# B&R Automation Studio project NAINV104C00R8L515F00 (part 18)

#### Act_Background.st
```iecst
(** 2020-10-05 **)
ACTION Act_Background: //For Standard Machines

	IF EDGEPOS(p_bManual) THEN

		fbBlink(bEn := FALSE);
		fbWarning(bEn := FALSE);

		bTLRed		:= FALSE;
		bTLAmber	:= TRUE;
		bTLGreen	:= FALSE;
		bBuzBeep	:= FALSE;

	ELSIF p_bManual THEN

		IF p_bErr = TRUE THEN

			fbBlink.tOnTm	:= p_tTLErrBlinkTm; //Error T#500ms (from NtParam)
			fbBlink.tOffTm	:= p_tTLErrBlinkTm; //Error T#500ms (from NtParam)

			fbWarning.tOnTm					:= p_tBuzErrOnTm; //Warn T#500ms (from NtParam)
			fbWarning.tOffTm				:= p_tBuzErrOnTm; //Warn T#500ms (from NtParam)
			fbWarning.tRstTm				:= p_tBuzErrRestTm; //Rest 5 seconds (from NtParam)
			fbWarning.usiOnCnt				:= p_usiBuzErrOnCntr; //Count 3 times (from NtParam)
			fbWarning.bStopAftRptSeqEn		:= p_bBuzErrStopSeqEn; //Enable Sequence Count (from NtParam)
			fbWarning.usiStopAftRptSeqCntr	:= p_usiBuzErrStopSeqCntr; //Sequence Counter  (from NtParam)

			fbBlink(bEn := TRUE);
			fbWarning(bEn := TRUE);

			bTLRed		:= fbBlink.bOut;
			bBuzBeep	:= (fbWarning.bOut) AND (p_bMuteBuz = FALSE);

			bManualErrOn := TRUE;

		ELSIF bManualErrOn THEN

			fbBlink(bEn := FALSE);
			fbWarning(bEn := FALSE);

			bTLRed		:= FALSE;
			bBuzBeep	:= FALSE;

			bManualErrOn := FALSE;

		END_IF

	ELSIF p_bManual = FALSE THEN

		bManualErrOn := FALSE;

		IF p_bStartup = TRUE THEN

			fbBlink(bEn := FALSE);
			fbWarning(bEn := FALSE);

			bTLRed		:= TRUE;
			bTLAmber	:= TRUE;
			bTLGreen	:= TRUE;
			bBuzBeep	:= FALSE;

		ELSIF p_bErr = TRUE THEN

			fbBlink.tOnTm	:= p_tTLErrBlinkTm; //Error T#500ms (from NtParam)
			fbBlink.tOffTm	:= p_tTLErrBlinkTm; //Error T#500ms (from NtParam)

			fbWarning.tOnTm					:= p_tBuzErrOnTm; //Warn T#500ms (from NtParam)
			fbWarning.tOffTm				:= p_tBuzErrOnTm; //Warn T#500ms (from NtParam)
			fbWarning.tRstTm				:= p_tBuzErrRestTm; //Rest 5 seconds (from NtParam)
			fbWarning.usiOnCnt				:= p_usiBuzErrOnCntr; //Count 3 times (from NtParam)
			fbWarning.bStopAftRptSeqEn		:= p_bBuzErrStopSeqEn; //Enable Sequence Count (from NtParam)
			fbWarning.usiStopAftRptSeqCntr	:= p_usiBuzErrStopSeqCntr; //Sequence Counter  (from NtParam)

			fbBlink(bEn := TRUE);
			fbWarning(bEn := TRUE);

			bTLRed		:= fbBlink.bOut;
			bTLAmber	:= FALSE;
			bTLGreen	:= FALSE;
			bBuzBeep	:= (fbWarning.bOut) AND (p_bMuteBuz = FALSE);

		ELSIF p_bErrNoBuz = TRUE THEN

			fbBlink.tOnTm	:= p_tTLErrBlinkTm;
			fbBlink.tOffTm	:= p_tTLErrBlinkTm;
			fbBlink(bEn := TRUE);
			fbWarning(bEn := FALSE);

			bTLRed		:= fbBlink.bOut;
			bTLAmber	:= FALSE;
			bTLGreen	:= FALSE;
			bBuzBeep	:= FALSE;

		ELSIF p_bWarning = TRUE THEN

			fbBlink.tOnTm	:= p_tTLWarnBlinkTm; //Warn T#500ms (from NtParam)
			fbBlink.tOffTm	:= p_tTLWarnBlinkTm; //Warn T#500ms (from NtParam)

			fbWarning.tOnTm					:= p_tBuzWarnOnTm; //Warn T#500ms (from NtParam)
			fbWarning.tOffTm				:= p_tBuzWarnOnTm; //Warn T#500ms (from NtParam)
			fbWarning.tRstTm				:= p_tBuzWarnRestTm; //Rest 5 seconds (from NtParam)
			fbWarning.usiOnCnt				:= p_usiBuzWarnOnCntr; //Count 3 times (from NtParam)
			fbWarning.bStopAftRptSeqEn		:= p_bBuzWarnStopSeqEn; //Enable Sequence Count (from NtParam)
			fbWarning.usiStopAftRptSeqCntr	:= p_usiBuzWarnStopSeqCntr; //Sequence Counter  (from NtParam)

			fbBlink(bEn := TRUE);
			fbWarning(bEn := TRUE);

			bTLRed		:= p_bStandby;
			bTLAmber	:= fbBlink.bOut;
			bTLGreen	:= p_bOps;
			bBuzBeep	:= fbWarning.bOut AND (p_bMuteBuz = FALSE);

		ELSIF p_bWarningNoBuz = TRUE THEN

			fbBlink.tOnTm	:= p_tTLWarnBlinkTm;
			fbBlink.tOffTm	:= p_tTLWarnBlinkTm;
			fbBlink(bEn := TRUE);
			fbWarning(bEn := FALSE);

			bTLRed		:= p_bStandby;
			bTLAmber	:= fbBlink.bOut;
			bTLGreen	:= p_bOps;
			bBuzBeep	:= FALSE;

		ELSIF p_bWarning1 = TRUE THEN

			fbBlink.tOnTm	:= p_tTLWarn1BlinkTm;
			fbBlink.tOffTm	:= p_tTLWarn1BlinkTm;

			fbWarning.tOnTm					:= p_tBuzWarn1OnTm; //Warn T#500ms (from NtParam)
			fbWarning.tOffTm				:= p_tBuzWarn1OnTm; //Warn T#500ms (from NtParam)
			fbWarning.tRstTm				:= p_tBuzWarn1RestTm; //Rest 5 seconds (from NtParam)
			fbWarning.usiOnCnt				:= p_usiBuzWarn1OnCntr; //Count 3 times (from NtParam)
			fbWarning.bStopAftRptSeqEn		:= p_bBuzWarn1StopSeqEn; //Enable Sequence Count (from NtParam)
			fbWarning.usiStopAftRptSeqCntr	:= p_usiBuzWarn1StopSeqCntr; //Sequence Counter  (from NtParam)

			fbBlink(bEn := TRUE);
			fbWarning(bEn := TRUE);

			bTLRed		:= p_bStandby;
			bTLAmber	:= fbBlink.bOut;
			bTLGreen	:= p_bOps;
			bBuzBeep	:= fbWarning.bOut AND (p_bMuteBuz = FALSE);

		ELSIF p_bWarning1NoBuz = TRUE THEN

			fbBlink.tOnTm	:= p_tTLWarn1BlinkTm;
			fbBlink.tOffTm	:= p_tTLWarn1BlinkTm;
			fbBlink(bEn := TRUE);
			fbWarning(bEn := FALSE);

			bTLRed		:= p_bStandby;
			bTLAmber	:= fbBlink.bOut;
			bTLGreen	:= p_bOps;
			bBuzBeep	:= FALSE;

		ELSIF p_bWarning2 = TRUE THEN

			fbBlink.tOnTm	:= p_tTLWarn2BlinkTm;
			fbBlink.tOffTm	:= p_tTLWarn2BlinkTm;

			fbWarning.tOnTm					:= p_tBuzWarn2OnTm; //Warn T#500ms (from NtParam)
			fbWarning.tOffTm				:= p_tBuzWarn2OnTm; //Warn T#500ms (from NtParam)
			fbWarning.tRstTm				:= p_tBuzWarn2RestTm; //Rest 5 seconds (from NtParam)
			fbWarning.usiOnCnt				:= p_usiBuzWarn2OnCntr; //Count 3 times (from NtParam)
			fbWarning.bStopAftRptSeqEn		:= p_bBuzWarn2StopSeqEn; //Enable Sequence Count (from NtParam)
			fbWarning.usiStopAftRptSeqCntr	:= p_usiBuzWarn2StopSeqCntr; //Sequence Counter  (from NtParam)

			fbBlink(bEn := TRUE);
			fbWarning(bEn := TRUE);

			bTLRed		:= p_bStandby;
			bTLAmber	:= fbBlink.bOut;
			bTLGreen	:= p_bOps;
			bBuzBeep	:= fbWarning.bOut AND (p_bMuteBuz = FALSE);

		ELSIF p_bWarning2NoBuz = TRUE THEN

			fbBlink.tOnTm	:= p_tTLWarn2BlinkTm;
			fbBlink.tOffTm	:= p_tTLWarn2BlinkTm;
			fbBlink(bEn := TRUE);
			fbWarning(bEn := FALSE);

			bTLRed		:= p_bStandby;
			bTLAmber	:= fbBlink.bOut;
			bTLGreen	:= p_bOps;
			bBuzBeep	:= FALSE;

		ELSIF p_bWarning3 = TRUE THEN

			fbBlink.tOnTm	:= p_tTLWarn3BlinkTm;
			fbBlink.tOffTm	:= p_tTLWarn3BlinkTm;

			fbWarning.tOnTm					:= p_tBuzWarn3OnTm; //Warn T#500ms (from NtParam)
			fbWarning.tOffTm				:= p_tBuzWarn3OnTm; //Warn T#500ms (from NtParam)
			fbWarning.tRstTm				:= p_tBuzWarn3RestTm; //Rest 5 seconds (from NtParam)
			fbWarning.usiOnCnt				:= p_usiBuzWarn3OnCntr; //Count 3 times (from NtParam)
			fbWarning.bStopAftRptSeqEn		:= p_bBuzWarn3StopSeqEn; //Enable Sequence Count (from NtParam)
			fbWarning.usiStopAftRptSeqCntr	:= p_usiBuzWarn3StopSeqCntr; //Sequence Counter  (from NtParam)

			fbBlink(bEn := TRUE);
			fbWarning(bEn := TRUE);

			bTLRed		:= p_bStandby;
			bTLAmber	:= fbBlink.bOut;
			bTLGreen	:= p_bOps;
			bBuzBeep	:= fbWarning.bOut AND (p_bMuteBuz = FALSE);

		ELSIF p_bWarning3NoBuz = TRUE THEN

			fbBlink.tOnTm	:= p_tTLWarn3BlinkTm;
			fbBlink.tOffTm	:= p_tTLWarn3BlinkTm;
			fbBlink(bEn := TRUE);
			fbWarning(bEn := FALSE);

			bTLRed		:= p_bStandby;
			bTLAmber	:= fbBlink.bOut;
			bTLGreen	:= p_bOps;
			bBuzBeep	:= FALSE;

		ELSIF p_bWarning4 = TRUE THEN

			fbBlink.tOnTm	:= p_tTLWarn4BlinkTm;
			fbBlink.tOffTm	:= p_tTLWarn4BlinkTm;

			fbWarning.tOnTm					:= p_tBuzWarn4OnTm; //Warn T#500ms (from NtParam)
			fbWarning.tOffTm				:= p_tBuzWarn4OnTm; //Warn T#500ms (from NtParam)
			fbWarning.tRstTm				:= p_tBuzWarn4RestTm; //Rest 5 seconds (from NtParam)
			fbWarning.usiOnCnt				:= p_usiBuzWarn4OnCntr; //Count 3 times (from NtParam)
			fbWarning.bStopAftRptSeqEn		:= p_bBuzWarn4StopSeqEn; //Enable Sequence Count (from NtParam)
			fbWarning.usiStopAftRptSeqCntr	:= p_usiBuzWarn4StopSeqCntr; //Sequence Counter  (from NtParam)

			fbBlink(bEn := TRUE);
			fbWarning(bEn := TRUE);

			bTLRed		:= p_bStandby;
			bTLAmber	:= fbBlink.bOut;
			bTLGreen	:= p_bOps;
			bBuzBeep	:= fbWarning.bOut AND (p_bMuteBuz = FALSE);

		ELSIF p_bWarning4NoBuz = TRUE THEN

			fbBlink.tOnTm	:= p_tTLWarn4BlinkTm;
			fbBlink.tOffTm	:= p_tTLWarn4BlinkTm;
			fbBlink(bEn := TRUE);
			fbWarning(bEn := FALSE);

			bTLRed		:= p_bStandby;
			bTLAmber	:= fbBlink.bOut;
			bTLGreen	:= p_bOps;
			bBuzBeep	:= FALSE;

		ELSIF p_bWarning5 = TRUE THEN

			fbBlink.tOnTm	:= p_tTLWarn5BlinkTm;
			fbBlink.tOffTm	:= p_tTLWarn5BlinkTm;

			fbWarning.tOnTm					:= p_tBuzWarn5OnTm; //Warn T#500ms (from NtParam)
			fbWarning.tOffTm				:= p_tBuzWarn5OnTm; //Warn T#500ms (from NtParam)
			fbWarning.tRstTm				:= p_tBuzWarn5RestTm; //Rest 5 seconds (from NtParam)
			fbWarning.usiOnCnt				:= p_usiBuzWarn5OnCntr; //Count 3 times (from NtParam)
			fbWarning.bStopAftRptSeqEn		:= p_bBuzWarn5StopSeqEn; //Enable Sequence Count (from NtParam)
			fbWarning.usiStopAftRptSeqCntr	:= p_usiBuzWarn5StopSeqCntr; //Sequence Counter  (from NtParam)

			fbBlink(bEn := TRUE);
			fbWarning(bEn := TRUE);

			bTLRed		:= p_bStandby;
			bTLAmber	:= fbBlink.bOut;
			bTLGreen	:= p_bOps;
			bBuzBeep	:= fbWarning.bOut AND (p_bMuteBuz = FALSE);

		ELSIF p_bWarning5NoBuz = TRUE THEN

			fbBlink.tOnTm	:= p_tTLWarn5BlinkTm;
			fbBlink.tOffTm	:= p_tTLWarn5BlinkTm;
			fbBlink(bEn := TRUE);
			fbWarning(bEn := FALSE);

			bTLRed		:= p_bStandby;
			bTLAmber	:= fbBlink.bOut;
			bTLGreen	:= p_bOps;
			bBuzBeep	:= FALSE;

		ELSIF p_bSeqStop = TRUE THEN

			fbBlink.tOnTm	:= tBlinkTm;
			fbBlink.tOffTm	:= tBlinkTm;
			fbBlink(bEn := TRUE);
			fbWarning(bEn := FALSE);

			bTLRed		:= fbBlink.bOut;
			bTLAmber	:= FALSE;
			bTLGreen	:= TRUE;
			bBuzBeep	:= FALSE;

		ELSIF p_bChgRcp = TRUE THEN

			fbBlink.tOnTm	:= p_tTLChgRcpBlinkTm;
			fbBlink.tOffTm	:= p_tTLChgRcpBlinkTm;
			fbBlink(bEn := TRUE);
			fbWarning(bEn := FALSE);

			IF EDGE(fbBlink.bOut) THEN
				IF bTLRed = TRUE THEN
					bTLRed		:= FALSE;
					bTLAmber	:= FALSE;
					bTLGreen	:= TRUE;
				ELSIF bTLAmber = TRUE THEN
					bTLRed		:= TRUE;
					bTLAmber	:= FALSE;
					bTLGreen	:= FALSE;
				ELSE
					bTLRed		:= FALSE;
					bTLAmber	:= TRUE;
					bTLGreen	:= FALSE;
				END_IF
			END_IF

			bBuzBeep	:= fbBlink.bOut AND (p_bMuteBuz = FALSE);

		ELSIF p_bStep = TRUE THEN

			fbBlink.tOnTm	:= tBlinkTm;
			fbBlink.tOffTm	:= tBlinkTm;
			fbBlink(bEn := TRUE);
			fbWarning(bEn := FALSE);

			bTLRed		:= FALSE;
			bTLAmber	:= FALSE;
			bTLGreen	:= fbBlink.bOut;
			bBuzBeep	:= FALSE;

		ELSIF p_bOps = TRUE THEN

			fbBlink(bEn := FALSE);
			fbWarning(bEn := FALSE);

			bTLRed		:= FALSE;
			bTLAmber	:= FALSE;
			bTLGreen	:= TRUE;
			bBuzBeep	:= FALSE;

		ELSIF p_bSimulation = TRUE THEN

			fbBlink.tOnTm	:= tBlinkTm;
			fbBlink.tOffTm	:= tBlinkTm;
			fbBlink(bEn := TRUE);
			fbWarning(bEn := FALSE);

			bTLRed		:= fbBlink.bOut;
			bTLAmber	:= fbBlink.bOut;
			bTLGreen	:= TRUE;
			bBuzBeep	:= FALSE;

		ELSIF p_bStandby = TRUE THEN

			fbBlink(bEn := FALSE);
			fbWarning(bEn := FALSE);

			bTLRed		:= TRUE;
			bTLAmber	:= FALSE;
			bTLGreen	:= FALSE;
			bBuzBeep	:= FALSE;

		ELSE

			fbBlink(bEn := FALSE);
			fbWarning(bEn := FALSE);

			bTLRed		:= FALSE;
			bTLAmber	:= FALSE;
			bTLGreen	:= FALSE;
			bBuzBeep	:= FALSE;

		END_IF

	END_IF

	IF p_bManual = FALSE AND p_bErr = FALSE THEN
		IF p_bTLAmberFlashEn THEN //Amber Flash 1 sec [Put Conditions in Act_Link.st]

			fbBlink1.tOnTm	:= p_tTLAmberBlinkTm; //T#500ms (from NtParam)
			fbBlink1.tOffTm	:= p_tTLAmberBlinkTm; //T#500ms (from NtParam)
			fbBlink1(bEn := TRUE);

			bTLAmber	:= fbBlink1.bOut;

		ELSE
			fbBlink1(bEn := FALSE);
		END_IF

		IF p_bTLRedFlashEn THEN //Red Flash 1 sec [Put Conditions in Act_Link.st]

			fbBlink2.tOnTm	:= p_tTLRedBlinkTm; //T#500ms (from NtParam)
			fbBlink2.tOffTm	:= p_tTLRedBlinkTm; //T#500ms (from NtParam)
			fbBlink2(bEn := TRUE);

			bTLRed		:= fbBlink2.bOut;
		ELSE
			fbBlink2(bEn := FALSE);
		END_IF

		IF p_bTLGreenFlashEn THEN //Green Flash 1 sec [Put Conditions in Act_Link.st]

			fbBlink3.tOnTm	:= p_tTLGreenBlinkTm; //T#500ms (from NtParam)
			fbBlink3.tOffTm	:= p_tTLGreenBlinkTm; //T#500ms (from NtParam)
			fbBlink3(bEn := TRUE);

			bTLGreen	:= fbBlink3.bOut;
		ELSE
			fbBlink3(bEn := FALSE);
		END_IF

		IF p_bBuzAlertEn = TRUE AND fbWarning.bEn=FALSE THEN

			fbWarning1.tOnTm				:= p_tBuzAlertOnTm;
			fbWarning1.tOffTm				:= p_tBuzAlertOnTm;
			fbWarning1.tRstTm				:= p_tBuzAlertRestTm;
			fbWarning1.usiOnCnt				:= p_usiBuzAlertOnCntr;
			fbWarning1.bStopAftRptSeqEn		:= p_bBuzAlertStopSeqEn; //Enable Sequence Count (from NtParam)
			fbWarning1.usiStopAftRptSeqCntr	:= p_usiBuzAlertStopSeqCntr; //Sequence Counter  (from NtParam)

			fbWarning1(bEn := TRUE);

			bBuzBeep	:= fbWarning1.bOut AND (p_bMuteBuz = FALSE);

		ELSE
			fbWarning1(bEn := FALSE);
		END_IF
	ELSE
		fbBlink1(bEn := FALSE);
		fbBlink2(bEn := FALSE);
		fbBlink3(bEn := FALSE);
		fbWarning1(bEn := FALSE);
	END_IF

	//Arrange p_bWarning according to the severity of the warning or info (Err is prioritized)
	IF p_bErr THEN
		usiWarnInfoStateNew	:= 1;
	ELSIF p_bWarning THEN
		usiWarnInfoStateNew	:= 2;
	ELSIF p_bWarning1 THEN
		usiWarnInfoStateNew	:= 3;
	ELSIF p_bWarning2 THEN
		usiWarnInfoStateNew	:= 4;
	ELSIF p_bWarning3 THEN
		usiWarnInfoStateNew	:= 5;
	ELSIF p_bWarning4 THEN
		usiWarnInfoStateNew	:= 6;
	ELSIF p_bWarning5 THEN
		usiWarnInfoStateNew	:= 7;
	ELSIF p_bBuzAlertEn AND fbWarning.bEn=FALSE THEN
		usiWarnInfoStateNew	:= 8;
	ELSE
		usiWarnInfoStateNew	:= 0;
	END_IF

	IF usiWarnInfoStateOld<>usiWarnInfoStateNew THEN
		usiWarnInfoStateOld:=usiWarnInfoStateNew;
		fbWarning(bEn := FALSE);
		fbWarning1(bEn := FALSE);
	END_IF

END_ACTION
```

#### Act_Background1.st
```iecst
(** 2020-10-05 **)
ACTION Act_Background1: //For Aptiv Machines

	IF EDGEPOS(p_bManual) THEN

		fbBlink(bEn := FALSE);
		fbWarning(bEn := FALSE);

		bTLRed		:= FALSE;
		bTLAmber	:= TRUE;
		bTLGreen	:= FALSE;
		bBuzBeep	:= FALSE;

	ELSIF p_bManual THEN

		IF p_bErr = TRUE THEN

			fbBlink.tOnTm	:= p_tTLErrBlinkTm; //Error T#500ms (from NtParam)
			fbBlink.tOffTm	:= p_tTLErrBlinkTm; //Error T#500ms (from NtParam)

			fbWarning.tOnTm					:= p_tBuzErrOnTm; //Warn T#500ms (from NtParam)
			fbWarning.tOffTm				:= p_tBuzErrOnTm; //Warn T#500ms (from NtParam)
			fbWarning.tRstTm				:= p_tBuzErrRestTm; //Rest 5 seconds (from NtParam)
			fbWarning.usiOnCnt				:= p_usiBuzErrOnCntr; //Count 3 times (from NtParam)
			fbWarning.bStopAftRptSeqEn		:= p_bBuzErrStopSeqEn; //Enable Sequence Count (from NtParam)
			fbWarning.usiStopAftRptSeqCntr	:= p_usiBuzErrStopSeqCntr; //Sequence Counter  (from NtParam)

			fbBlink(bEn := TRUE);
			fbWarning(bEn := TRUE);

			bTLRed		:= TRUE;
			bBuzBeep	:= (fbWarning.bOut) AND (p_bMuteBuz = FALSE);

			bManualErrOn := TRUE;

		ELSIF bManualErrOn THEN

			fbBlink(bEn := FALSE);
			fbWarning(bEn := FALSE);

			bTLRed		:= FALSE;
			bBuzBeep	:= FALSE;

			bManualErrOn := FALSE;

		END_IF

	ELSIF p_bManual = FALSE THEN

		bManualErrOn := FALSE;

		IF p_bStartup = TRUE THEN

			fbBlink(bEn := FALSE);
			fbWarning(bEn := FALSE);

			bTLRed		:= TRUE;
			bTLAmber	:= TRUE;
			bTLGreen	:= TRUE;
			bBuzBeep	:= FALSE;

		ELSIF p_bCoverSwitchSig = FALSE THEN

			fbBlink.tOnTm	:= p_tTLErrBlinkTm;
			fbBlink.tOffTm	:= p_tTLErrBlinkTm;
			fbBlink(bEn := TRUE);
			fbWarning(bEn := FALSE);

			bTLRed		:= fbBlink.bOut;
			bTLAmber	:= FALSE;
			bTLGreen	:= FALSE;
			bBuzBeep	:= (fbBlink.bOut) AND (p_bMuteBuz = FALSE);

		ELSIF p_bErr = TRUE THEN

			fbBlink.tOnTm	:= p_tTLErrBlinkTm; //Error T#500ms (from NtParam)
			fbBlink.tOffTm	:= p_tTLErrBlinkTm; //Error T#500ms (from NtParam)

			fbWarning.tOnTm					:= p_tBuzErrOnTm; //Warn T#500ms (from NtParam)
			fbWarning.tOffTm				:= p_tBuzErrOnTm; //Warn T#500ms (from NtParam)
			fbWarning.tRstTm				:= p_tBuzErrRestTm; //Rest 5 seconds (from NtParam)
			fbWarning.usiOnCnt				:= p_usiBuzErrOnCntr; //Count 3 times (from NtParam)
			fbWarning.bStopAftRptSeqEn		:= p_bBuzErrStopSeqEn; //Enable Sequence Count (from NtParam)
			fbWarning.usiStopAftRptSeqCntr	:= p_usiBuzErrStopSeqCntr; //Sequence Counter  (from NtParam)

			fbBlink(bEn := TRUE);
			fbWarning(bEn := TRUE);

			bTLRed		:= TRUE;
			bTLAmber	:= FALSE;
			bTLGreen	:= FALSE;
			bBuzBeep	:= (fbWarning.bOut) AND (p_bMuteBuz = FALSE);

		ELSIF p_bErrNoBuz = TRUE THEN

			fbBlink.tOnTm	:= p_tTLErrBlinkTm;
			fbBlink.tOffTm	:= p_tTLErrBlinkTm;
			fbBlink(bEn := TRUE);
			fbWarning(bEn := FALSE);

			bTLRed		:= fbBlink.bOut;
			bTLAmber	:= FALSE;
			bTLGreen	:= FALSE;
			bBuzBeep	:= FALSE;

		ELSIF p_bWarning = TRUE THEN

			fbBlink.tOnTm	:= p_tTLWarnBlinkTm; //Warn T#500ms (from NtParam)
			fbBlink.tOffTm	:= p_tTLWarnBlinkTm; //Warn T#500ms (from NtParam)

			fbWarning.tOnTm					:= p_tBuzWarnOnTm; //Warn T#500ms (from NtParam)
			fbWarning.tOffTm				:= p_tBuzWarnOnTm; //Warn T#500ms (from NtParam)
			fbWarning.tRstTm				:= p_tBuzWarnRestTm; //Rest 5 seconds (from NtParam)
			fbWarning.usiOnCnt				:= p_usiBuzWarnOnCntr; //Count 3 times (from NtParam)
			fbWarning.bStopAftRptSeqEn		:= p_bBuzWarnStopSeqEn; //Enable Sequence Count (from NtParam)
			fbWarning.usiStopAftRptSeqCntr	:= p_usiBuzWarnStopSeqCntr; //Sequence Counter  (from NtParam)

			fbBlink(bEn := TRUE);
			fbWarning(bEn := TRUE);

			bTLRed		:= FALSE;
			bTLAmber	:= fbBlink.bOut;
			bTLGreen	:= FALSE;
			bBuzBeep	:= fbWarning.bOut AND (p_bMuteBuz = FALSE);

		ELSIF p_bWarningNoBuz = TRUE THEN

			fbBlink.tOnTm	:= p_tTLWarnBlinkTm;
			fbBlink.tOffTm	:= p_tTLWarnBlinkTm;
			fbBlink(bEn := TRUE);
			fbWarning(bEn := FALSE);

			bTLRed		:= FALSE;
			bTLAmber	:= fbBlink.bOut;
			bTLGreen	:= FALSE;
			bBuzBeep	:= FALSE;

		ELSIF p_bWarning1 = TRUE THEN

			fbBlink.tOnTm	:= p_tTLWarn1BlinkTm;
			fbBlink.tOffTm	:= p_tTLWarn1BlinkTm;

			fbWarning.tOnTm					:= p_tBuzWarn1OnTm; //Warn T#500ms (from NtParam)
			fbWarning.tOffTm				:= p_tBuzWarn1OnTm; //Warn T#500ms (from NtParam)
			fbWarning.tRstTm				:= p_tBuzWarn1RestTm; //Rest 5 seconds (from NtParam)
			fbWarning.usiOnCnt				:= p_usiBuzWarn1OnCntr; //Count 3 times (from NtParam)
			fbWarning.bStopAftRptSeqEn		:= p_bBuzWarn1StopSeqEn; //Enable Sequence Count (from NtParam)
			fbWarning.usiStopAftRptSeqCntr	:= p_usiBuzWarn1StopSeqCntr; //Sequence Counter  (from NtParam)

			fbBlink(bEn := TRUE);
			fbWarning(bEn := TRUE);

			bTLRed		:= p_bStandby;
			bTLAmber	:= fbBlink.bOut;
			bTLGreen	:= p_bOps;
			bBuzBeep	:= fbWarning.bOut AND (p_bMuteBuz = FALSE);

		ELSIF p_bWarning1NoBuz = TRUE THEN

			fbBlink.tOnTm	:= p_tTLWarn1BlinkTm;
			fbBlink.tOffTm	:= p_tTLWarn1BlinkTm;
			fbBlink(bEn := TRUE);
			fbWarning(bEn := FALSE);

			bTLRed		:= p_bStandby;
			bTLAmber	:= fbBlink.bOut;
			bTLGreen	:= p_bOps;
			bBuzBeep	:= FALSE;

		ELSIF p_bWarning2 = TRUE THEN

			fbBlink.tOnTm	:= p_tTLWarn2BlinkTm;
			fbBlink.tOffTm	:= p_tTLWarn2BlinkTm;

			fbWarning.tOnTm					:= p_tBuzWarn2OnTm; //Warn T#500ms (from NtParam)
			fbWarning.tOffTm				:= p_tBuzWarn2OnTm; //Warn T#500ms (from NtParam)
			fbWarning.tRstTm				:= p_tBuzWarn2RestTm; //Rest 5 seconds (from NtParam)
			fbWarning.usiOnCnt				:= p_usiBuzWarn2OnCntr; //Count 3 times (from NtParam)
			fbWarning.bStopAftRptSeqEn		:= p_bBuzWarn2StopSeqEn; //Enable Sequence Count (from NtParam)
			fbWarning.usiStopAftRptSeqCntr	:= p_usiBuzWarn2StopSeqCntr; //Sequence Counter  (from NtParam)

			fbBlink(bEn := TRUE);
			fbWarning(bEn := TRUE);

			bTLRed		:= p_bStandby;
			bTLAmber	:= fbBlink.bOut;
			bTLGreen	:= p_bOps;
			bBuzBeep	:= fbWarning.bOut AND (p_bMuteBuz = FALSE);

		ELSIF p_bWarning2NoBuz = TRUE THEN

			fbBlink.tOnTm	:= p_tTLWarn2BlinkTm;
			fbBlink.tOffTm	:= p_tTLWarn2BlinkTm;
			fbBlink(bEn := TRUE);
			fbWarning(bEn := FALSE);

			bTLRed		:= p_bStandby;
			bTLAmber	:= fbBlink.bOut;
			bTLGreen	:= p_bOps;
			bBuzBeep	:= FALSE;

		ELSIF p_bWarning3 = TRUE THEN

			fbBlink.tOnTm	:= p_tTLWarn3BlinkTm;
			fbBlink.tOffTm	:= p_tTLWarn3BlinkTm;

			fbWarning.tOnTm					:= p_tBuzWarn3OnTm; //Warn T#500ms (from NtParam)
			fbWarning.tOffTm				:= p_tBuzWarn3OnTm; //Warn T#500ms (from NtParam)
			fbWarning.tRstTm				:= p_tBuzWarn3RestTm; //Rest 5 seconds (from NtParam)
			fbWarning.usiOnCnt				:= p_usiBuzWarn3OnCntr; //Count 3 times (from NtParam)
			fbWarning.bStopAftRptSeqEn		:= p_bBuzWarn3StopSeqEn; //Enable Sequence Count (from NtParam)
			fbWarning.usiStopAftRptSeqCntr	:= p_usiBuzWarn3StopSeqCntr; //Sequence Counter  (from NtParam)

			fbBlink(bEn := TRUE);
			fbWarning(bEn := TRUE);

			bTLRed		:= p_bStandby;
			bTLAmber	:= fbBlink.bOut;
			bTLGreen	:= p_bOps;
			bBuzBeep	:= fbWarning.bOut AND (p_bMuteBuz = FALSE);

		ELSIF p_bWarning3NoBuz = TRUE THEN

			fbBlink.tOnTm	:= p_tTLWarn3BlinkTm;
			fbBlink.tOffTm	:= p_tTLWarn3BlinkTm;
			fbBlink(bEn := TRUE);
			fbWarning(bEn := FALSE);

			bTLRed		:= p_bStandby;
			bTLAmber	:= fbBlink.bOut;
			bTLGreen	:= p_bOps;
			bBuzBeep	:= FALSE;

		ELSIF p_bWarning4 = TRUE THEN

			fbBlink.tOnTm	:= p_tTLWarn4BlinkTm;
			fbBlink.tOffTm	:= p_tTLWarn4BlinkTm;

			fbWarning.tOnTm					:= p_tBuzWarn4OnTm; //Warn T#500ms (from NtParam)
			fbWarning.tOffTm				:= p_tBuzWarn4OnTm; //Warn T#500ms (from NtParam)
			fbWarning.tRstTm				:= p_tBuzWarn4RestTm; //Rest 5 seconds (from NtParam)
			fbWarning.usiOnCnt				:= p_usiBuzWarn4OnCntr; //Count 3 times (from NtParam)
			fbWarning.bStopAftRptSeqEn		:= p_bBuzWarn4StopSeqEn; //Enable Sequence Count (from NtParam)
			fbWarning.usiStopAftRptSeqCntr	:= p_usiBuzWarn4StopSeqCntr; //Sequence Counter  (from NtParam)

			fbBlink(bEn := TRUE);
			fbWarning(bEn := TRUE);

			bTLRed		:= p_bStandby;
			bTLAmber	:= fbBlink.bOut;
			bTLGreen	:= p_bOps;
			bBuzBeep	:= fbWarning.bOut AND (p_bMuteBuz = FALSE);

		ELSIF p_bWarning4NoBuz = TRUE THEN

			fbBlink.tOnTm	:= p_tTLWarn4BlinkTm;
			fbBlink.tOffTm	:= p_tTLWarn4BlinkTm;
			fbBlink(bEn := TRUE);
			fbWarning(bEn := FALSE);

			bTLRed		:= p_bStandby;
			bTLAmber	:= fbBlink.bOut;
			bTLGreen	:= p_bOps;
			bBuzBeep	:= FALSE;

		ELSIF p_bWarning5 = TRUE THEN

			fbBlink.tOnTm	:= p_tTLWarn5BlinkTm;
			fbBlink.tOffTm	:= p_tTLWarn5BlinkTm;

			fbWarning.tOnTm					:= p_tBuzWarn5OnTm; //Warn T#500ms (from NtParam)
			fbWarning.tOffTm				:= p_tBuzWarn5OnTm; //Warn T#500ms (from NtParam)
			fbWarning.tRstTm				:= p_tBuzWarn5RestTm; //Rest 5 seconds (from NtParam)
			fbWarning.usiOnCnt				:= p_usiBuzWarn5OnCntr; //Count 3 times (from NtParam)
			fbWarning.bStopAftRptSeqEn		:= p_bBuzWarn5StopSeqEn; //Enable Sequence Count (from NtParam)
			fbWarning.usiStopAftRptSeqCntr	:= p_usiBuzWarn5StopSeqCntr; //Sequence Counter  (from NtParam)

			fbBlink(bEn := TRUE);
			fbWarning(bEn := TRUE);

			bTLRed		:= p_bStandby;
			bTLAmber	:= fbBlink.bOut;
			bTLGreen	:= p_bOps;
			bBuzBeep	:= fbWarning.bOut AND (p_bMuteBuz = FALSE);

		ELSIF p_bWarning5NoBuz = TRUE THEN

			fbBlink.tOnTm	:= p_tTLWarn5BlinkTm;
			fbBlink.tOffTm	:= p_tTLWarn5BlinkTm;
			fbBlink(bEn := TRUE);
			fbWarning(bEn := FALSE);

			bTLRed		:= p_bStandby;
			bTLAmber	:= fbBlink.bOut;
			bTLGreen	:= p_bOps;
			bBuzBeep	:= FALSE;

		ELSIF p_bSeqStop = TRUE THEN

			fbBlink.tOnTm	:= tBlinkTm;
			fbBlink.tOffTm	:= tBlinkTm;
			fbBlink(bEn := TRUE);
			fbWarning(bEn := FALSE);

			bTLRed		:= FALSE;
			bTLAmber	:= FALSE;
			bTLGreen	:= fbBlink.bOut;
			bBuzBeep	:= FALSE;

		ELSIF p_bChgRcp = TRUE THEN

			fbBlink.tOnTm	:= p_tTLChgRcpBlinkTm;
			fbBlink.tOffTm	:= p_tTLChgRcpBlinkTm;
			fbBlink(bEn := TRUE);
			fbWarning(bEn := FALSE);

			IF EDGE(fbBlink.bOut) THEN
				IF bTLRed = TRUE THEN
					bTLRed		:= FALSE;
					bTLAmber	:= FALSE;
					bTLGreen	:= TRUE;
				ELSIF bTLAmber = TRUE THEN
					bTLRed		:= TRUE;
					bTLAmber	:= FALSE;
					bTLGreen	:= FALSE;
				ELSE
					bTLRed		:= FALSE;
					bTLAmber	:= TRUE;
					bTLGreen	:= FALSE;
				END_IF
			END_IF

			bBuzBeep	:= fbBlink.bOut AND (p_bMuteBuz = FALSE);

		ELSIF p_bStep = TRUE THEN

			fbBlink.tOnTm	:= tBlinkTm;
			fbBlink.tOffTm	:= tBlinkTm;
			fbBlink(bEn := TRUE);
			fbWarning(bEn := FALSE);

			bTLRed		:= FALSE;
			bTLAmber	:= FALSE;
			bTLGreen	:= fbBlink.bOut;
			bBuzBeep	:= FALSE;

		ELSIF p_bOps = TRUE THEN

			fbBlink(bEn := FALSE);
			fbWarning(bEn := FALSE);

			bTLRed		:= FALSE;
			bTLAmber	:= FALSE;
			bTLGreen	:= TRUE;
			bBuzBeep	:= FALSE;

		ELSIF p_bSimulation = TRUE THEN

			fbBlink.tOnTm	:= tBlinkTm;
			fbBlink.tOffTm	:= tBlinkTm;
			fbBlink(bEn := TRUE);
			fbWarning(bEn := FALSE);

			bTLRed		:= fbBlink.bOut;
			bTLAmber	:= fbBlink.bOut;
			bTLGreen	:= TRUE;
			bBuzBeep	:= FALSE;

		ELSIF p_bStandby = TRUE THEN

			fbBlink(bEn := FALSE);
			fbWarning(bEn := FALSE);

			bTLRed		:= FALSE;
			bTLAmber	:= TRUE;
			bTLGreen	:= FALSE;
			bBuzBeep	:= FALSE;

		ELSE

			fbBlink(bEn := FALSE);
			fbWarning(bEn := FALSE);

			bTLRed		:= FALSE;
			bTLAmber	:= FALSE;
			bTLGreen	:= FALSE;
			bBuzBeep	:= FALSE;

		END_IF

	END_IF

	IF p_bManual = FALSE AND p_bErr = FALSE THEN
		IF p_bTLAmberFlashEn THEN //Amber Flash 1 sec [Put Conditions in Act_Link.st]

			fbBlink1.tOnTm	:= p_tTLAmberBlinkTm; //T#500ms (from NtParam)
			fbBlink1.tOffTm	:= p_tTLAmberBlinkTm; //T#500ms (from NtParam)
			fbBlink1(bEn := TRUE);

			bTLAmber	:= fbBlink1.bOut;

		ELSE
			fbBlink1(bEn := FALSE);
		END_IF

		IF p_bTLRedFlashEn THEN //Red Flash 1 sec [Put Conditions in Act_Link.st]

			fbBlink2.tOnTm	:= p_tTLRedBlinkTm; //T#500ms (from NtParam)
			fbBlink2.tOffTm	:= p_tTLRedBlinkTm; //T#500ms (from NtParam)
			fbBlink2(bEn := TRUE);

			bTLRed		:= fbBlink2.bOut;
		ELSE
			fbBlink2(bEn := FALSE);
		END_IF

		IF p_bTLGreenFlashEn THEN //Green Flash 1 sec [Put Conditions in Act_Link.st]

			fbBlink3.tOnTm	:= p_tTLGreenBlinkTm; //T#500ms (from NtParam)
			fbBlink3.tOffTm	:= p_tTLGreenBlinkTm; //T#500ms (from NtParam)
			fbBlink3(bEn := TRUE);

			bTLGreen	:= fbBlink3.bOut;
		ELSE
			fbBlink3(bEn := FALSE);
		END_IF

		IF p_bBuzAlertEn = TRUE AND fbWarning.bEn=FALSE THEN

			fbWarning1.tOnTm				:= p_tBuzAlertOnTm;
			fbWarning1.tOffTm				:= p_tBuzAlertOnTm;
			fbWarning1.tRstTm				:= p_tBuzAlertRestTm;
			fbWarning1.usiOnCnt				:= p_usiBuzAlertOnCntr;
			fbWarning1.bStopAftRptSeqEn		:= p_bBuzAlertStopSeqEn; //Enable Sequence Count (from NtParam)
			fbWarning1.usiStopAftRptSeqCntr	:= p_usiBuzAlertStopSeqCntr; //Sequence Counter  (from NtParam)

			fbWarning1(bEn := TRUE);

			bBuzBeep	:= fbWarning1.bOut AND (p_bMuteBuz = FALSE);

		ELSE
			fbWarning1(bEn := FALSE);
		END_IF
	ELSE
		fbBlink1(bEn := FALSE);
		fbBlink2(bEn := FALSE);
		fbBlink3(bEn := FALSE);
		fbWarning1(bEn := FALSE);
	END_IF

	//Arrange p_bWarning according to the severity of the warning or info (Err is prioritized)
	IF p_bErr THEN
		usiWarnInfoStateNew	:= 1;
	ELSIF p_bWarning THEN
		usiWarnInfoStateNew	:= 2;
	ELSIF p_bWarning1 THEN
		usiWarnInfoStateNew	:= 3;
	ELSIF p_bWarning2 THEN
		usiWarnInfoStateNew	:= 4;
	ELSIF p_bWarning3 THEN
		usiWarnInfoStateNew	:= 5;
	ELSIF p_bWarning4 THEN
		usiWarnInfoStateNew	:= 6;
	ELSIF p_bWarning5 THEN
		usiWarnInfoStateNew	:= 7;
	ELSIF p_bBuzAlertEn AND fbWarning.bEn=FALSE THEN
		usiWarnInfoStateNew	:= 8;
	ELSE
		usiWarnInfoStateNew	:= 0;
	END_IF

	IF usiWarnInfoStateOld<>usiWarnInfoStateNew THEN
		usiWarnInfoStateOld:=usiWarnInfoStateNew;
		fbWarning(bEn := FALSE);
		fbWarning1(bEn := FALSE);
	END_IF

END_ACTION
```

#### Act_Background2.st
```iecst
(** 2020-10-05 **)
ACTION Act_Background2: //For MEK machines

	IF EDGEPOS(p_bManual) THEN

		fbBlink(bEn := FALSE);
		fbWarning(bEn := FALSE);

		bTLRed		:= FALSE;
		bTLAmber	:= TRUE;
		bTLGreen	:= FALSE;
		bBuzBeep	:= FALSE;

	ELSIF p_bManual THEN

		IF p_bErr = TRUE THEN

			fbBlink.tOnTm	:= p_tTLErrBlinkTm; //Error T#500ms (from NtParam)
			fbBlink.tOffTm	:= p_tTLErrBlinkTm; //Error T#500ms (from NtParam)

			fbWarning.tOnTm					:= p_tBuzErrOnTm; //Warn T#500ms (from NtParam)
			fbWarning.tOffTm				:= p_tBuzErrOnTm; //Warn T#500ms (from NtParam)
			fbWarning.tRstTm				:= p_tBuzErrRestTm; //Rest 5 seconds (from NtParam)
			fbWarning.usiOnCnt				:= p_usiBuzErrOnCntr; //Count 3 times (from NtParam)
			fbWarning.bStopAftRptSeqEn		:= p_bBuzErrStopSeqEn; //Enable Sequence Count (from NtParam)
			fbWarning.usiStopAftRptSeqCntr	:= p_usiBuzErrStopSeqCntr; //Sequence Counter  (from NtParam)

			fbBlink(bEn := TRUE);
			fbWarning(bEn := TRUE);

			bTLRed		:= fbBlink.bOut;
			bBuzBeep	:= (fbWarning.bOut) AND (p_bMuteBuz = FALSE);

			bManualErrOn := TRUE;

		ELSIF bManualErrOn THEN

			fbBlink(bEn := FALSE);
			fbWarning(bEn := FALSE);

			bTLRed		:= FALSE;
			bBuzBeep	:= FALSE;

			bManualErrOn := FALSE;

		END_IF

	ELSIF p_bManual = FALSE THEN

		bManualErrOn := FALSE;

		IF p_bStartup = TRUE THEN

			fbBlink(bEn := FALSE);
			fbWarning(bEn := FALSE);

			bTLRed		:= TRUE;
			bTLAmber	:= TRUE;
			bTLGreen	:= TRUE;
			bBuzBeep	:= FALSE;

		ELSIF p_bErr = TRUE THEN

			fbBlink.tOnTm	:= p_tTLErrBlinkTm; //Error T#500ms (from NtParam)
			fbBlink.tOffTm	:= p_tTLErrBlinkTm; //Error T#500ms (from NtParam)

			fbWarning.tOnTm					:= p_tBuzErrOnTm; //Warn T#500ms (from NtParam)
			fbWarning.tOffTm				:= p_tBuzErrOnTm; //Warn T#500ms (from NtParam)
			fbWarning.tRstTm				:= p_tBuzErrRestTm; //Rest 5 seconds (from NtParam)
			fbWarning.usiOnCnt				:= p_usiBuzErrOnCntr; //Count 3 times (from NtParam)
			fbWarning.bStopAftRptSeqEn		:= p_bBuzErrStopSeqEn; //Enable Sequence Count (from NtParam)
			fbWarning.usiStopAftRptSeqCntr	:= p_usiBuzErrStopSeqCntr; //Sequence Counter  (from NtParam)

			fbBlink(bEn := TRUE);
			fbWarning(bEn := TRUE);

			bTLRed		:= fbBlink.bOut;
			bTLAmber	:= FALSE;
			bTLGreen	:= FALSE;
			bBuzBeep	:= (fbWarning.bOut) AND (p_bMuteBuz = FALSE);

		ELSIF p_bErrNoBuz = TRUE THEN

			fbBlink.tOnTm	:= p_tTLErrBlinkTm;
			fbBlink.tOffTm	:= p_tTLErrBlinkTm;
			fbBlink(bEn := TRUE);
			fbWarning(bEn := FALSE);

			bTLRed		:= fbBlink.bOut;
			bTLAmber	:= FALSE;
			bTLGreen	:= FALSE;
			bBuzBeep	:= FALSE;

		ELSIF p_bOps = TRUE AND p_bAOIErrSig = TRUE AND p_bAOIOriginSig = FALSE THEN

			fbBlink.tOnTm	:= p_tTLErrBlinkTm;
			fbBlink.tOffTm	:= p_tTLErrBlinkTm;
			fbBlink(bEn := TRUE);
			fbWarning(bEn := FALSE);

			bTLRed		:= fbBlink.bOut;
			bTLAmber	:= FALSE;
			bTLGreen	:= FALSE;
			bBuzBeep	:= (fbBlink.bOut) AND (p_bMuteBuz = FALSE);

		ELSIF p_bOps = TRUE AND p_bAOIErrSig = TRUE AND p_bAOIOriginSig = TRUE THEN

			fbBlink.tOnTm	:= p_tTLErrBlinkTm;
			fbBlink.tOffTm	:= p_tTLErrBlinkTm;
			fbBlink(bEn := TRUE);
			fbWarning(bEn := FALSE);

			bTLRed		:= fbBlink.bOut;
			bTLAmber	:= FALSE;
			bTLGreen	:= TRUE;
			bBuzBeep	:= (fbBlink.bOut) AND (p_bMuteBuz = FALSE);

		ELSIF p_bWarning = TRUE THEN

			fbBlink.tOnTm	:= p_tTLWarnBlinkTm; //Warn T#500ms (from NtParam)
			fbBlink.tOffTm	:= p_tTLWarnBlinkTm; //Warn T#500ms (from NtParam)

			fbWarning.tOnTm					:= p_tBuzWarnOnTm; //Warn T#500ms (from NtParam)
			fbWarning.tOffTm				:= p_tBuzWarnOnTm; //Warn T#500ms (from NtParam)
			fbWarning.tRstTm				:= p_tBuzWarnRestTm; //Rest 5 seconds (from NtParam)
			fbWarning.usiOnCnt				:= p_usiBuzWarnOnCntr; //Count 3 times (from NtParam)
			fbWarning.bStopAftRptSeqEn		:= p_bBuzWarnStopSeqEn; //Enable Sequence Count (from NtParam)
			fbWarning.usiStopAftRptSeqCntr	:= p_usiBuzWarnStopSeqCntr; //Sequence Counter  (from NtParam)

			fbBlink(bEn := TRUE);
			fbWarning(bEn := TRUE);

			bTLRed		:= p_bStandby;
			bTLAmber	:= fbBlink.bOut;
			bTLGreen	:= p_bOps;
			bBuzBeep	:= fbWarning.bOut AND (p_bMuteBuz = FALSE);

		ELSIF p_bWarningNoBuz = TRUE THEN

			fbBlink.tOnTm	:= p_tTLWarnBlinkTm;
			fbBlink.tOffTm	:= p_tTLWarnBlinkTm;
			fbBlink(bEn := TRUE);
			fbWarning(bEn := FALSE);

			bTLRed		:= p_bStandby;
			bTLAmber	:= fbBlink.bOut;
			bTLGreen	:= p_bOps;
			bBuzBeep	:= FALSE;

		ELSIF p_bWarning1 = TRUE THEN

			fbBlink.tOnTm	:= p_tTLWarn1BlinkTm;
			fbBlink.tOffTm	:= p_tTLWarn1BlinkTm;

			fbWarning.tOnTm					:= p_tBuzWarn1OnTm; //Warn T#500ms (from NtParam)
			fbWarning.tOffTm				:= p_tBuzWarn1OnTm; //Warn T#500ms (from NtParam)
			fbWarning.tRstTm				:= p_tBuzWarn1RestTm; //Rest 5 seconds (from NtParam)
			fbWarning.usiOnCnt				:= p_usiBuzWarn1OnCntr; //Count 3 times (from NtParam)
			fbWarning.bStopAftRptSeqEn		:= p_bBuzWarn1StopSeqEn; //Enable Sequence Count (from NtParam)
			fbWarning.usiStopAftRptSeqCntr	:= p_usiBuzWarn1StopSeqCntr; //Sequence Counter  (from NtParam)

			fbBlink(bEn := TRUE);
			fbWarning(bEn := TRUE);

			bTLRed		:= p_bStandby;
			bTLAmber	:= fbBlink.bOut;
			bTLGreen	:= p_bOps;
			bBuzBeep	:= fbWarning.bOut AND (p_bMuteBuz = FALSE);

		ELSIF p_bWarning1NoBuz = TRUE THEN

			fbBlink.tOnTm	:= p_tTLWarn1BlinkTm;
			fbBlink.tOffTm	:= p_tTLWarn1BlinkTm;
			fbBlink(bEn := TRUE);
			fbWarning(bEn := FALSE);

			bTLRed		:= p_bStandby;
			bTLAmber	:= fbBlink.bOut;
			bTLGreen	:= p_bOps;
			bBuzBeep	:= FALSE;

		ELSIF p_bWarning2 = TRUE THEN

			fbBlink.tOnTm	:= p_tTLWarn2BlinkTm;
			fbBlink.tOffTm	:= p_tTLWarn2BlinkTm;

			fbWarning.tOnTm					:= p_tBuzWarn2OnTm; //Warn T#500ms (from NtParam)
			fbWarning.tOffTm				:= p_tBuzWarn2OnTm; //Warn T#500ms (from NtParam)
			fbWarning.tRstTm				:= p_tBuzWarn2RestTm; //Rest 5 seconds (from NtParam)
			fbWarning.usiOnCnt				:= p_usiBuzWarn2OnCntr; //Count 3 times (from NtParam)
			fbWarning.bStopAftRptSeqEn		:= p_bBuzWarn2StopSeqEn; //Enable Sequence Count (from NtParam)
			fbWarning.usiStopAftRptSeqCntr	:= p_usiBuzWarn2StopSeqCntr; //Sequence Counter  (from NtParam)

			fbBlink(bEn := TRUE);
			fbWarning(bEn := TRUE);

			bTLRed		:= p_bStandby;
			bTLAmber	:= fbBlink.bOut;
			bTLGreen	:= p_bOps;
			bBuzBeep	:= fbWarning.bOut AND (p_bMuteBuz = FALSE);

		ELSIF p_bWarning2NoBuz = TRUE THEN

			fbBlink.tOnTm	:= p_tTLWarn2BlinkTm;
			fbBlink.tOffTm	:= p_tTLWarn2BlinkTm;
			fbBlink(bEn := TRUE);
			fbWarning(bEn := FALSE);

			bTLRed		:= p_bStandby;
			bTLAmber	:= fbBlink.bOut;
			bTLGreen	:= p_bOps;
			bBuzBeep	:= FALSE;

		ELSIF p_bWarning3 = TRUE THEN

			fbBlink.tOnTm	:= p_tTLWarn3BlinkTm;
			fbBlink.tOffTm	:= p_tTLWarn3BlinkTm;

			fbWarning.tOnTm					:= p_tBuzWarn3OnTm; //Warn T#500ms (from NtParam)
			fbWarning.tOffTm				:= p_tBuzWarn3OnTm; //Warn T#500ms (from NtParam)
			fbWarning.tRstTm				:= p_tBuzWarn3RestTm; //Rest 5 seconds (from NtParam)
			fbWarning.usiOnCnt				:= p_usiBuzWarn3OnCntr; //Count 3 times (from NtParam)
			fbWarning.bStopAftRptSeqEn		:= p_bBuzWarn3StopSeqEn; //Enable Sequence Count (from NtParam)
			fbWarning.usiStopAftRptSeqCntr	:= p_usiBuzWarn3StopSeqCntr; //Sequence Counter  (from NtParam)

			fbBlink(bEn := TRUE);
			fbWarning(bEn := TRUE);

			bTLRed		:= p_bStandby;
			bTLAmber	:= fbBlink.bOut;
			bTLGreen	:= p_bOps;
			bBuzBeep	:= fbWarning.bOut AND (p_bMuteBuz = FALSE);

		ELSIF p_bWarning3NoBuz = TRUE THEN

			fbBlink.tOnTm	:= p_tTLWarn3BlinkTm;
			fbBlink.tOffTm	:= p_tTLWarn3BlinkTm;
			fbBlink(bEn := TRUE);
			fbWarning(bEn := FALSE);

			bTLRed		:= p_bStandby;
			bTLAmber	:= fbBlink.bOut;
			bTLGreen	:= p_bOps;
			bBuzBeep	:= FALSE;

		ELSIF p_bWarning4 = TRUE THEN

			fbBlink.tOnTm	:= p_tTLWarn4BlinkTm;
			fbBlink.tOffTm	:= p_tTLWarn4BlinkTm;

			fbWarning.tOnTm					:= p_tBuzWarn4OnTm; //Warn T#500ms (from NtParam)
			fbWarning.tOffTm				:= p_tBuzWarn4OnTm; //Warn T#500ms (from NtParam)
			fbWarning.tRstTm				:= p_tBuzWarn4RestTm; //Rest 5 seconds (from NtParam)
			fbWarning.usiOnCnt				:= p_usiBuzWarn4OnCntr; //Count 3 times (from NtParam)
			fbWarning.bStopAftRptSeqEn		:= p_bBuzWarn4StopSeqEn; //Enable Sequence Count (from NtParam)
			fbWarning.usiStopAftRptSeqCntr	:= p_usiBuzWarn4StopSeqCntr; //Sequence Counter  (from NtParam)

			fbBlink(bEn := TRUE);
			fbWarning(bEn := TRUE);

			bTLRed		:= p_bStandby;
			bTLAmber	:= fbBlink.bOut;
			bTLGreen	:= p_bOps;
			bBuzBeep	:= fbWarning.bOut AND (p_bMuteBuz = FALSE);

		ELSIF p_bWarning4NoBuz = TRUE THEN

			fbBlink.tOnTm	:= p_tTLWarn4BlinkTm;
			fbBlink.tOffTm	:= p_tTLWarn4BlinkTm;
			fbBlink(bEn := TRUE);
			fbWarning(bEn := FALSE);

			bTLRed		:= p_bStandby;
			bTLAmber	:= fbBlink.bOut;
			bTLGreen	:= p_bOps;
			bBuzBeep	:= FALSE;

		ELSIF p_bWarning5 = TRUE THEN

			fbBlink.tOnTm	:= p_tTLWarn5BlinkTm;
			fbBlink.tOffTm	:= p_tTLWarn5BlinkTm;

			fbWarning.tOnTm					:= p_tBuzWarn5OnTm; //Warn T#500ms (from NtParam)
			fbWarning.tOffTm				:= p_tBuzWarn5OnTm; //Warn T#500ms (from NtParam)
			fbWarning.tRstTm				:= p_tBuzWarn5RestTm; //Rest 5 seconds (from NtParam)
			fbWarning.usiOnCnt				:= p_usiBuzWarn5OnCntr; //Count 3 times (from NtParam)
			fbWarning.bStopAftRptSeqEn		:= p_bBuzWarn5StopSeqEn; //Enable Sequence Count (from NtParam)
			fbWarning.usiStopAftRptSeqCntr	:= p_usiBuzWarn5StopSeqCntr; //Sequence Counter  (from NtParam)

			fbBlink(bEn := TRUE);
			fbWarning(bEn := TRUE);

			bTLRed		:= p_bStandby;
			bTLAmber	:= fbBlink.bOut;
			bTLGreen	:= p_bOps;
			bBuzBeep	:= fbWarning.bOut AND (p_bMuteBuz = FALSE);

		ELSIF p_bWarning5NoBuz = TRUE THEN

			fbBlink.tOnTm	:= p_tTLWarn5BlinkTm;
			fbBlink.tOffTm	:= p_tTLWarn5BlinkTm;
			fbBlink(bEn := TRUE);
			fbWarning(bEn := FALSE);

			bTLRed		:= p_bStandby;
			bTLAmber	:= fbBlink.bOut;
			bTLGreen	:= p_bOps;
			bBuzBeep	:= FALSE;

		ELSIF p_bSeqStop = TRUE THEN

			fbBlink.tOnTm	:= tBlinkTm;
			fbBlink.tOffTm	:= tBlinkTm;
			fbBlink(bEn := TRUE);
			fbWarning(bEn := FALSE);

			bTLRed		:= fbBlink.bOut;
			bTLAmber	:= FALSE;
			bTLGreen	:= TRUE;
			bBuzBeep	:= FALSE;

		ELSIF p_bChgRcp = TRUE THEN

			fbBlink.tOnTm	:= p_tTLChgRcpBlinkTm;
			fbBlink.tOffTm	:= p_tTLChgRcpBlinkTm;
			fbBlink(bEn := TRUE);
			fbWarning(bEn := FALSE);

			IF EDGE(fbBlink.bOut) THEN
				IF bTLRed = TRUE THEN
					bTLRed		:= FALSE;
					bTLAmber	:= FALSE;
					bTLGreen	:= TRUE;
				ELSIF bTLAmber = TRUE THEN
					bTLRed		:= TRUE;
					bTLAmber	:= FALSE;
					bTLGreen	:= FALSE;
				ELSE
					bTLRed		:= FALSE;
					bTLAmber	:= TRUE;
					bTLGreen	:= FALSE;
				END_IF
			END_IF

			bBuzBeep	:= fbBlink.bOut AND (p_bMuteBuz = FALSE);

		ELSIF p_bStep = TRUE THEN

			fbBlink.tOnTm	:= tBlinkTm;
			fbBlink.tOffTm	:= tBlinkTm;
			fbBlink(bEn := TRUE);
			fbWarning(bEn := FALSE);

			bTLRed		:= FALSE;
			bTLAmber	:= FALSE;
			bTLGreen	:= fbBlink.bOut;
			bBuzBeep	:= FALSE;

		ELSIF p_bOps = TRUE THEN

			fbBlink(bEn := FALSE);
			fbWarning(bEn := FALSE);

			bTLRed		:= FALSE;
			bTLAmber	:= FALSE;
			bTLGreen	:= TRUE;
			bBuzBeep	:= FALSE;

		ELSIF p_bSimulation = TRUE THEN

			fbBlink.tOnTm	:= tBlinkTm;
			fbBlink.tOffTm	:= tBlinkTm;
			fbBlink(bEn := TRUE);
			fbWarning(bEn := FALSE);

			bTLRed		:= fbBlink.bOut;
			bTLAmber	:= fbBlink.bOut;
			bTLGreen	:= TRUE;
			bBuzBeep	:= FALSE;

		ELSIF p_bStandby = TRUE THEN

			fbBlink(bEn := FALSE);
			fbWarning(bEn := FALSE);

			bTLRed		:= TRUE;
			bTLAmber	:= FALSE;
			bTLGreen	:= FALSE;
			bBuzBeep	:= FALSE;

		ELSE

			fbBlink(bEn := FALSE);
			fbWarning(bEn := FALSE);

			bTLRed		:= FALSE;
			bTLAmber	:= FALSE;
			bTLGreen	:= FALSE;
			bBuzBeep	:= FALSE;

		END_IF

	END_IF

	IF p_bManual = FALSE AND p_bErr = FALSE THEN
		IF p_bTLAmberFlashEn THEN //Amber Flash 1 sec [Put Conditions in Act_Link.st]

			fbBlink1.tOnTm	:= p_tTLAmberBlinkTm; //T#500ms (from NtParam)
			fbBlink1.tOffTm	:= p_tTLAmberBlinkTm; //T#500ms (from NtParam)
			fbBlink1(bEn := TRUE);

			bTLAmber	:= fbBlink1.bOut;

		ELSE
			fbBlink1(bEn := FALSE);
		END_IF

		IF p_bTLRedFlashEn THEN //Red Flash 1 sec [Put Conditions in Act_Link.st]

			fbBlink2.tOnTm	:= p_tTLRedBlinkTm; //T#500ms (from NtParam)
			fbBlink2.tOffTm	:= p_tTLRedBlinkTm; //T#500ms (from NtParam)
			fbBlink2(bEn := TRUE);

			bTLRed		:= fbBlink2.bOut;
		ELSE
			fbBlink2(bEn := FALSE);
		END_IF

		IF p_bTLGreenFlashEn THEN //Green Flash 1 sec [Put Conditions in Act_Link.st]

			fbBlink3.tOnTm	:= p_tTLGreenBlinkTm; //T#500ms (from NtParam)
			fbBlink3.tOffTm	:= p_tTLGreenBlinkTm; //T#500ms (from NtParam)
			fbBlink3(bEn := TRUE);

			bTLGreen	:= fbBlink3.bOut;
		ELSE
			fbBlink3(bEn := FALSE);
		END_IF

		IF p_bBuzAlertEn = TRUE AND fbWarning.bEn=FALSE THEN

			fbWarning1.tOnTm				:= p_tBuzAlertOnTm;
			fbWarning1.tOffTm				:= p_tBuzAlertOnTm;
			fbWarning1.tRstTm				:= p_tBuzAlertRestTm;
			fbWarning1.usiOnCnt				:= p_usiBuzAlertOnCntr;
			fbWarning1.bStopAftRptSeqEn		:= p_bBuzAlertStopSeqEn; //Enable Sequence Count (from NtParam)
			fbWarning1.usiStopAftRptSeqCntr	:= p_usiBuzAlertStopSeqCntr; //Sequence Counter  (from NtParam)

			fbWarning1(bEn := TRUE);

			bBuzBeep	:= fbWarning1.bOut AND (p_bMuteBuz = FALSE);

		ELSE
			fbWarning1(bEn := FALSE);
		END_IF
	ELSE
		fbBlink1(bEn := FALSE);
		fbBlink2(bEn := FALSE);
		fbBlink3(bEn := FALSE);
		fbWarning1(bEn := FALSE);
	END_IF

	//Arrange p_bWarning according to the severity of the warning or info (Err is prioritized)
	IF p_bErr THEN
		usiWarnInfoStateNew	:= 1;
	ELSIF p_bWarning THEN
		usiWarnInfoStateNew	:= 2;
	ELSIF p_bWarning1 THEN
		usiWarnInfoStateNew	:= 3;
	ELSIF p_bWarning2 THEN
		usiWarnInfoStateNew	:= 4;
	ELSIF p_bWarning3 THEN
		usiWarnInfoStateNew	:= 5;
	ELSIF p_bWarning4 THEN
		usiWarnInfoStateNew	:= 6;
	ELSIF p_bWarning5 THEN
		usiWarnInfoStateNew	:= 7;
	ELSIF p_bBuzAlertEn AND fbWarning.bEn=FALSE THEN
		usiWarnInfoStateNew	:= 8;
	ELSE
		usiWarnInfoStateNew	:= 0;
	END_IF

	IF usiWarnInfoStateOld<>usiWarnInfoStateNew THEN
		usiWarnInfoStateOld:=usiWarnInfoStateNew;
		fbWarning(bEn := FALSE);
		fbWarning1(bEn := FALSE);
	END_IF

END_ACTION
```

#### Act_Background3.st
```iecst
(** 2020-10-05 **)
ACTION Act_Background3: //For BHTC Machines

	IF EDGEPOS(p_bManual) THEN

		fbBlink(bEn := FALSE);
		fbWarning(bEn := FALSE);

		bTLRed		:= FALSE;
		bTLAmber	:= FALSE;
		bTLWhite	:= TRUE;
		bTLGreen	:= FALSE;
		bBuzBeep	:= FALSE;

	ELSIF p_bManual THEN

		IF p_bErr = TRUE THEN

			fbBlink.tOnTm	:= p_tTLErrBlinkTm; //Error T#500ms (from NtParam)
			fbBlink.tOffTm	:= p_tTLErrBlinkTm; //Error T#500ms (from NtParam)

			fbWarning.tOnTm					:= p_tBuzErrOnTm; //Warn T#500ms (from NtParam)
			fbWarning.tOffTm				:= p_tBuzErrOnTm; //Warn T#500ms (from NtParam)
			fbWarning.tRstTm				:= p_tBuzErrRestTm; //Rest 5 seconds (from NtParam)
			fbWarning.usiOnCnt				:= p_usiBuzErrOnCntr; //Count 3 times (from NtParam)
			fbWarning.bStopAftRptSeqEn		:= p_bBuzErrStopSeqEn; //Enable Sequence Count (from NtParam)
			fbWarning.usiStopAftRptSeqCntr	:= p_usiBuzErrStopSeqCntr; //Sequence Counter  (from NtParam)

			fbBlink(bEn := TRUE);
			fbWarning(bEn := TRUE);

			bTLAmber	:= fbBlink.bOut;
			bBuzBeep	:= (fbWarning.bOut) AND (p_bMuteBuz = FALSE);

			bManualErrOn := TRUE;

		ELSIF bManualErrOn THEN

			fbBlink(bEn := FALSE);
			fbWarning(bEn := FALSE);

			bTLAmber	:= FALSE;
			bBuzBeep	:= FALSE;

			bManualErrOn := FALSE;

		END_IF

	ELSIF p_bManual = FALSE THEN

		bManualErrOn := FALSE;

		IF p_bStartup = TRUE THEN //Startup, 3 colour ON

			fbBlink(bEn := FALSE);
			fbWarning(bEn := FALSE);

			bTLBlue		:= TRUE;
			bTLAmber	:= TRUE;
			bTLWhite	:= TRUE;
			bTLGreen	:= TRUE;
			bBuzBeep	:= FALSE;

		ELSIF p_bErr = TRUE THEN //Machine Error,Green TL Off, Red TL Blink

			fbBlink.tOnTm	:= p_tTLErrBlinkTm; //Error T#500ms (from NtParam)
			fbBlink.tOffTm	:= p_tTLErrBlinkTm; //Error T#500ms (from NtParam)

			fbWarning.tOnTm					:= p_tBuzErrOnTm; //Warn T#500ms (from NtParam)
			fbWarning.tOffTm				:= p_tBuzErrOnTm; //Warn T#500ms (from NtParam)
			fbWarning.tRstTm				:= p_tBuzErrRestTm; //Rest 5 seconds (from NtParam)
			fbWarning.usiOnCnt				:= p_usiBuzErrOnCntr; //Count 3 times (from NtParam)
			fbWarning.bStopAftRptSeqEn		:= p_bBuzErrStopSeqEn; //Enable Sequence Count (from NtParam)
			fbWarning.usiStopAftRptSeqCntr	:= p_usiBuzErrStopSeqCntr; //Sequence Counter  (from NtParam)

			fbBlink(bEn := TRUE);
			fbWarning(bEn := TRUE);

			bTLBlue		:= FALSE;
			bTLAmber	:= fbBlink.bOut;
			bTLWhite	:= FALSE;
			bTLGreen	:= FALSE;
			bBuzBeep	:= fbWarning.bOut AND (p_bMuteBuz = FALSE);

		ELSIF p_bErrNoBuz = TRUE THEN //not used (Machine Error With No Buz)

			fbBlink.tOnTm	:= p_tTLErrBlinkTm; //Error T#500ms, not used (from NtParam)
			fbBlink.tOffTm	:= p_tTLErrBlinkTm; //Error T#500ms, not used (from NtParam)
			fbBlink(bEn := TRUE);
			fbWarning(bEn := FALSE);

			bTLBlue		:= FALSE;
			bTLAmber	:= fbBlink.bOut;
			bTLWhite	:= FALSE;
			bTLGreen	:= FALSE;
			bBuzBeep	:= FALSE;

		ELSIF p_bWarning = TRUE THEN //Warning or AlarmInfo; [Put Conditions in Act_Link.st]

			fbBlink.tOnTm	:= p_tTLWarnBlinkTm; //Warn T#500ms (from NtParam)
			fbBlink.tOffTm	:= p_tTLWarnBlinkTm; //Warn T#500ms (from NtParam)

			fbWarning.tOnTm					:= p_tBuzWarnOnTm; //Warn T#500ms (from NtParam)
			fbWarning.tOffTm				:= p_tBuzWarnOnTm; //Warn T#500ms (from NtParam)
			fbWarning.tRstTm				:= p_tBuzWarnRestTm; //Rest 5 seconds (from NtParam)
			fbWarning.usiOnCnt				:= p_usiBuzWarnOnCntr; //Count 3 times (from NtParam)
			fbWarning.bStopAftRptSeqEn		:= p_bBuzWarnStopSeqEn; //Enable Sequence Count (from NtParam)
			fbWarning.usiStopAftRptSeqCntr	:= p_usiBuzWarnStopSeqCntr; //Sequence Counter  (from NtParam)

			fbBlink(bEn := TRUE);
			fbWarning(bEn := TRUE);

			bTLBlue		:= FALSE;
			bTLAmber	:= p_bStandby; //[p_bStandby ACCESS p_OpsStatusStop], [p_OpsStatusStop	:= ADR(bStatusStop);]
			bTLWhite	:= fbBlink.bOut;
			bTLGreen	:= p_bOps; //[p_bOps ACCESS p_OpsStatusRun],  [p_OpsStatusRun	:= ADR(bStatusRun)];
			bBuzBeep	:= fbWarning.bOut AND (p_bMuteBuz = FALSE);

		ELSIF p_bWarningNoBuz = TRUE THEN //not used

			fbBlink.tOnTm	:= p_tTLWarnBlinkTm;
			fbBlink.tOffTm	:= p_tTLWarnBlinkTm;
			fbBlink(bEn := TRUE);
			fbWarning(bEn := FALSE);

			bTLBlue		:= FALSE;
			bTLAmber	:= p_bStandby;
			bTLWhite	:= fbBlink.bOut;
			bTLGreen	:= p_bOps;
			bBuzBeep	:= FALSE;

		ELSIF p_bWarning1 = TRUE THEN //not used

			fbBlink.tOnTm	:= p_tTLWarn1BlinkTm;
			fbBlink.tOffTm	:= p_tTLWarn1BlinkTm;

			fbWarning.tOnTm					:= p_tBuzWarn1OnTm; //Warn T#500ms (from NtParam)
			fbWarning.tOffTm				:= p_tBuzWarn1OnTm; //Warn T#500ms (from NtParam)
			fbWarning.tRstTm				:= p_tBuzWarn1RestTm; //Rest 5 seconds (from NtParam)
			fbWarning.usiOnCnt				:= p_usiBuzWarn1OnCntr; //Count 3 times (from NtParam)
			fbWarning.bStopAftRptSeqEn		:= p_bBuzWarn1StopSeqEn; //Enable Sequence Count (from NtParam)
			fbWarning.usiStopAftRptSeqCntr	:= p_usiBuzWarn1StopSeqCntr; //Sequence Counter  (from NtParam)

			fbBlink(bEn := TRUE);
			fbWarning(bEn := TRUE);

			bTLBlue		:= FALSE;
			bTLAmber	:= p_bStandby;
			bTLWhite	:= fbBlink.bOut;
			bTLGreen	:= p_bOps;
			bBuzBeep	:= fbWarning.bOut AND (p_bMuteBuz = FALSE);

		ELSIF p_bWarning1NoBuz = TRUE THEN //not used

			fbBlink.tOnTm	:= p_tTLWarn1BlinkTm;
			fbBlink.tOffTm	:= p_tTLWarn1BlinkTm;
			fbBlink(bEn := TRUE);
			fbWarning(bEn := FALSE);

			bTLBlue		:= FALSE;
			bTLAmber	:= p_bStandby;
			bTLWhite	:= fbBlink.bOut;
			bTLGreen	:= p_bOps;
			bBuzBeep	:= FALSE;

		ELSIF p_bWarning2 = TRUE THEN //not used

			fbBlink.tOnTm	:= p_tTLWarn2BlinkTm;
			fbBlink.tOffTm	:= p_tTLWarn2BlinkTm;

			fbWarning.tOnTm					:= p_tBuzWarn2OnTm; //Warn T#500ms (from NtParam)
			fbWarning.tOffTm				:= p_tBuzWarn2OnTm; //Warn T#500ms (from NtParam)
			fbWarning.tRstTm				:= p_tBuzWarn2RestTm; //Rest 5 seconds (from NtParam)
			fbWarning.usiOnCnt				:= p_usiBuzWarn2OnCntr; //Count 3 times (from NtParam)
			fbWarning.bStopAftRptSeqEn		:= p_bBuzWarn2StopSeqEn; //Enable Sequence Count (from NtParam)
			fbWarning.usiStopAftRptSeqCntr	:= p_usiBuzWarn2StopSeqCntr; //Sequence Counter  (from NtParam)

			fbBlink(bEn := TRUE);
			fbWarning(bEn := TRUE);

			bTLBlue		:= FALSE;
			bTLAmber	:= p_bStandby;
			bTLWhite	:= fbBlink.bOut;
			bTLGreen	:= p_bOps;
			bBuzBeep	:= fbWarning.bOut AND (p_bMuteBuz = FALSE);

		ELSIF p_bWarning2NoBuz = TRUE THEN //not used

			fbBlink.tOnTm	:= p_tTLWarn2BlinkTm;
			fbBlink.tOffTm	:= p_tTLWarn2BlinkTm;
			fbBlink(bEn := TRUE);
			fbWarning(bEn := FALSE);

			bTLBlue		:= FALSE;
			bTLAmber	:= p_bStandby;
			bTLWhite	:= fbBlink.bOut;
			bTLGreen	:= p_bOps;
			bBuzBeep	:= FALSE;

		ELSIF p_bWarning3 = TRUE THEN //not used

			fbBlink.tOnTm	:= p_tTLWarn3BlinkTm;
			fbBlink.tOffTm	:= p_tTLWarn3BlinkTm;

			fbWarning.tOnTm					:= p_tBuzWarn3OnTm; //Warn T#500ms (from NtParam)
			fbWarning.tOffTm				:= p_tBuzWarn3OnTm; //Warn T#500ms (from NtParam)
			fbWarning.tRstTm				:= p_tBuzWarn3RestTm; //Rest 5 seconds (from NtParam)
			fbWarning.usiOnCnt				:= p_usiBuzWarn3OnCntr; //Count 3 times (from NtParam)
			fbWarning.bStopAftRptSeqEn		:= p_bBuzWarn3StopSeqEn; //Enable Sequence Count (from NtParam)
			fbWarning.usiStopAftRptSeqCntr	:= p_usiBuzWarn3StopSeqCntr; //Sequence Counter  (from NtParam)

			fbBlink(bEn := TRUE);
			fbWarning(bEn := TRUE);

			bTLBlue		:= FALSE;
			bTLAmber	:= p_bStandby;
			bTLWhite	:= fbBlink.bOut;
			bTLGreen	:= p_bOps;
			bBuzBeep	:= fbWarning.bOut AND (p_bMuteBuz = FALSE);

		ELSIF p_bWarning3NoBuz = TRUE THEN //not used

			fbBlink.tOnTm	:= p_tTLWarn3BlinkTm;
			fbBlink.tOffTm	:= p_tTLWarn3BlinkTm;
			fbBlink(bEn := TRUE);
			fbWarning(bEn := FALSE);

			bTLBlue		:= FALSE;
			bTLAmber	:= p_bStandby;
			bTLWhite	:= fbBlink.bOut;
			bTLGreen	:= p_bOps;
			bBuzBeep	:= FALSE;

		ELSIF p_bWarning4 = TRUE THEN //not used

			fbBlink.tOnTm	:= p_tTLWarn4BlinkTm;
			fbBlink.tOffTm	:= p_tTLWarn4BlinkTm;

			fbWarning.tOnTm					:= p_tBuzWarn4OnTm; //Warn T#500ms (from NtParam)
			fbWarning.tOffTm				:= p_tBuzWarn4OnTm; //Warn T#500ms (from NtParam)
			fbWarning.tRstTm				:= p_tBuzWarn4RestTm; //Rest 5 seconds (from NtParam)
			fbWarning.usiOnCnt				:= p_usiBuzWarn4OnCntr; //Count 3 times (from NtParam)
			fbWarning.bStopAftRptSeqEn		:= p_bBuzWarn4StopSeqEn; //Enable Sequence Count (from NtParam)
			fbWarning.usiStopAftRptSeqCntr	:= p_usiBuzWarn4StopSeqCntr; //Sequence Counter  (from NtParam)

			fbBlink(bEn := TRUE);
			fbWarning(bEn := TRUE);

			bTLBlue		:= FALSE;
			bTLAmber	:= p_bStandby;
			bTLWhite	:= fbBlink.bOut;
			bTLGreen	:= p_bOps;
			bBuzBeep	:= fbWarning.bOut AND (p_bMuteBuz = FALSE);

		ELSIF p_bWarning4NoBuz = TRUE THEN //not used

			fbBlink.tOnTm	:= p_tTLWarn4BlinkTm;
			fbBlink.tOffTm	:= p_tTLWarn4BlinkTm;
			fbBlink(bEn := TRUE);
			fbWarning(bEn := FALSE);

			bTLBlue		:= FALSE;
			bTLAmber	:= p_bStandby;
			bTLWhite	:= fbBlink.bOut;
			bTLGreen	:= p_bOps;
			bBuzBeep	:= FALSE;

		ELSIF p_bWarning5 = TRUE THEN //not used

			fbBlink.tOnTm	:= p_tTLWarn5BlinkTm;
			fbBlink.tOffTm	:= p_tTLWarn5BlinkTm;

			fbWarning.tOnTm					:= p_tBuzWarn5OnTm; //Warn T#500ms (from NtParam)
			fbWarning.tOffTm				:= p_tBuzWarn5OnTm; //Warn T#500ms (from NtParam)
			fbWarning.tRstTm				:= p_tBuzWarn5RestTm; //Rest 5 seconds (from NtParam)
			fbWarning.usiOnCnt				:= p_usiBuzWarn5OnCntr; //Count 3 times (from NtParam)
			fbWarning.bStopAftRptSeqEn		:= p_bBuzWarn5StopSeqEn; //Enable Sequence Count (from NtParam)
			fbWarning.usiStopAftRptSeqCntr	:= p_usiBuzWarn5StopSeqCntr; //Sequence Counter  (from NtParam)

			fbBlink(bEn := TRUE);
			fbWarning(bEn := TRUE);

			bTLBlue		:= FALSE;
			bTLAmber	:= p_bStandby;
			bTLWhite	:= fbBlink.bOut;
			bTLGreen	:= p_bOps;
			bBuzBeep	:= fbWarning.bOut AND (p_bMuteBuz = FALSE);

		ELSIF p_bWarning5NoBuz = TRUE THEN //not used

			fbBlink.tOnTm	:= p_tTLWarn5BlinkTm;
			fbBlink.tOffTm	:= p_tTLWarn5BlinkTm;
			fbBlink(bEn := TRUE);
			fbWarning(bEn := FALSE);

			bTLBlue		:= FALSE;
			bTLAmber	:= p_bStandby;
			bTLWhite	:= fbBlink.bOut;
			bTLGreen	:= p_bOps;
			bBuzBeep	:= FALSE;

		ELSIF p_bSeqStop = TRUE THEN //[p_bSeqStop ACCESS p_OpsStatusCycleStop] ,[p_OpsStatusCycleStop	:= ADR(bStatusCycleStop);]

			fbBlink.tOnTm	:= tBlinkTm; //Local T#500ms
			fbBlink.tOffTm	:= tBlinkTm; //Local T#500ms
			fbBlink(bEn := TRUE);
			fbWarning(bEn := FALSE);

			bTLBlue		:= FALSE;
			bTLAmber	:= fbBlink.bOut;
			bTLWhite	:= FALSE;
			bTLGreen	:= TRUE;
			bBuzBeep	:= FALSE;

		ELSIF p_bChgRcp = TRUE THEN //Change Rcp, Disco Light, not used

			fbBlink.tOnTm	:= p_tTLChgRcpBlinkTm; //Chg Rcp T#500ms (from NtParam)
			fbBlink.tOffTm	:= p_tTLChgRcpBlinkTm; //Chg Rcp T#500ms (from NtParam)
			fbBlink(bEn := TRUE);
			fbWarning(bEn := FALSE);

			IF EDGE(fbBlink.bOut) THEN
				IF bTLAmber = TRUE THEN
					bTLAmber	:= FALSE;
					bTLWhite	:= FALSE;
					bTLGreen	:= TRUE;
				ELSIF bTLWhite = TRUE THEN
					bTLAmber	:= TRUE;
					bTLWhite	:= FALSE;
					bTLGreen	:= FALSE;
				ELSE
					bTLAmber	:= FALSE;
					bTLWhite	:= TRUE;
					bTLGreen	:= FALSE;
				END_IF
			END_IF

			bBuzBeep	:= fbBlink.bOut AND (p_bMuteBuz = FALSE);

		ELSIF p_bStep = TRUE THEN //not used, [p_bStep ACCESS p_OpsStatusStep], [p_OpsStatusStep	:= ADR(bStatusStep);]

			fbBlink.tOnTm	:= tBlinkTm;
			fbBlink.tOffTm	:= tBlinkTm;
			fbBlink(bEn := TRUE);
			fbWarning(bEn := FALSE);

			bTLBlue		:= FALSE;
			bTLAmber	:= FALSE;
			bTLWhite	:= FALSE;
			bTLGreen	:= fbBlink.bOut;
			bBuzBeep	:= FALSE;

		ELSIF p_bOps = TRUE THEN //Auto Mode, Green TL only

			fbBlink(bEn := FALSE);
			fbWarning(bEn := FALSE);

			bTLRed		:= FALSE;
			bTLAmber	:= FALSE;
			bTLGreen	:= TRUE;
			bBuzBeep	:= FALSE;

		ELSIF p_bSimulation = TRUE THEN //For simulation

			fbBlink.tOnTm	:= tBlinkTm;
			fbBlink.tOffTm	:= tBlinkTm;
			fbBlink(bEn := TRUE);
			fbWarning(bEn := FALSE);

			bTLBlue		:= fbBlink.bOut;
			bTLAmber	:= fbBlink.bOut;
			bTLWhite	:= fbBlink.bOut;
			bTLGreen	:= TRUE;
			bBuzBeep	:= FALSE;

		ELSIF p_bStandby = TRUE THEN //Stop Mode, On Red TL only

			fbBlink(bEn := FALSE);
			fbWarning(bEn := FALSE);

			bTLBlue		:= FALSE;
			bTLAmber	:= TRUE;
			bTLWhite	:= FALSE;
			bTLGreen	:= FALSE;
			bBuzBeep	:= FALSE;

		ELSE //Resest if nothing else

			fbBlink(bEn := FALSE);
			fbWarning(bEn := FALSE);

			bTLBlue		:= FALSE;
			bTLAmber	:= FALSE;
			bTLWhite	:= FALSE;
			bTLGreen	:= FALSE;
			bBuzBeep	:= FALSE;

		END_IF

	END_IF

	IF p_bManual = FALSE AND p_bErr = FALSE THEN
		IF p_bTLAmberFlashEn THEN //Amber Flash 1 sec [Put Conditions in Act_Link.st]

			fbBlink1.tOnTm	:= p_tTLAmberBlinkTm; //T#500ms (from NtParam)
			fbBlink1.tOffTm	:= p_tTLAmberBlinkTm; //T#500ms (from NtParam)
			fbBlink1(bEn := TRUE);

			bTLAmber	:= fbBlink1.bOut;

		ELSE
			fbBlink1(bEn := FALSE);
		END_IF

		IF p_bTLWhiteFlashEn THEN //White Flash 1 sec [Put Conditions in Act_Link.st]

			fbBlink2.tOnTm	:= p_tTLWhiteBlinkTm; //T#500ms (from NtParam)
			fbBlink2.tOffTm	:= p_tTLWhiteBlinkTm; //T#500ms (from NtParam)
			fbBlink2(bEn := TRUE);

			bTLWhite		:= fbBlink2.bOut;
		ELSE
			fbBlink2(bEn := FALSE);
		END_IF

		IF p_bTLGreenFlashEn THEN //Green Flash 1 sec [Put Conditions in Act_Link.st]

			fbBlink3.tOnTm	:= p_tTLGreenBlinkTm; //T#500ms (from NtParam)
			fbBlink3.tOffTm	:= p_tTLGreenBlinkTm; //T#500ms (from NtParam)
			fbBlink3(bEn := TRUE);

			bTLGreen	:= fbBlink3.bOut;
		ELSE
			fbBlink3(bEn := FALSE);
		END_IF

		IF p_bTLBlueFlashEn THEN //Blue Flash 1 sec [Put Conditions in Act_Link.st]

			fbBlink4.tOnTm	:= p_tTLBlueBlinkTm; //T#500ms (from NtParam)
			fbBlink4.tOffTm	:= p_tTLBlueBlinkTm; //T#500ms (from NtParam)
			fbBlink4(bEn := TRUE);

			bTLGreen	:= fbBlink4.bOut;
		ELSE
			fbBlink4(bEn := FALSE);
		END_IF

		IF p_bBuzAlertEn = TRUE AND fbWarning.bEn=FALSE THEN

			fbWarning1.tOnTm				:= p_tBuzAlertOnTm;
			fbWarning1.tOffTm				:= p_tBuzAlertOnTm;
			fbWarning1.tRstTm				:= p_tBuzAlertRestTm;
			fbWarning1.usiOnCnt				:= p_usiBuzAlertOnCntr;
			fbWarning1.bStopAftRptSeqEn		:= p_bBuzAlertStopSeqEn; //Enable Sequence Count (from NtParam)
			fbWarning1.usiStopAftRptSeqCntr	:= p_usiBuzAlertStopSeqCntr; //Sequence Counter  (from NtParam)

			fbWarning1(bEn := TRUE);

			bBuzBeep	:= fbWarning1.bOut AND (p_bMuteBuz = FALSE);

		ELSE
			fbWarning1(bEn := FALSE);
		END_IF
	ELSE
		fbBlink1(bEn := FALSE);
		fbBlink2(bEn := FALSE);
		fbBlink3(bEn := FALSE);
		fbBlink4(bEn := FALSE);
		fbWarning1(bEn := FALSE);
	END_IF

	//Arrange p_bWarning according to the severity of the warning or info (Err is prioritized)
	IF p_bErr THEN
		usiWarnInfoStateNew	:= 1;
	ELSIF p_bWarning THEN
		usiWarnInfoStateNew	:= 2;
	ELSIF p_bWarning1 THEN
		usiWarnInfoStateNew	:= 3;
	ELSIF p_bWarning2 THEN
		usiWarnInfoStateNew	:= 4;
	ELSIF p_bWarning3 THEN
		usiWarnInfoStateNew	:= 5;
	ELSIF p_bWarning4 THEN
		usiWarnInfoStateNew	:= 6;
	ELSIF p_bWarning5 THEN
		usiWarnInfoStateNew	:= 7;
	ELSIF p_bBuzAlertEn AND fbWarning.bEn=FALSE THEN
		usiWarnInfoStateNew	:= 8;
	ELSE
		usiWarnInfoStateNew	:= 0;
	END_IF

	IF usiWarnInfoStateOld<>usiWarnInfoStateNew THEN
		usiWarnInfoStateOld:=usiWarnInfoStateNew;
		fbWarning(bEn := FALSE);
		fbWarning1(bEn := FALSE);
	END_IF

END_ACTION
```

#### InputRef.var - Do Not Change!!!
```iecst
(*2020-03-16*)
(**)
(*General*)
VAR
	p_eAct : REFERENCE TO eTLBuzAction;
END_VAR
(**)
(*Configuration*)
VAR
	p_bManual : REFERENCE TO BOOL;
	p_bStartup : REFERENCE TO BOOL;
	p_bErr : REFERENCE TO BOOL;
	p_bErrNoBuz : REFERENCE TO BOOL;
	p_bWarning : REFERENCE TO BOOL;
	p_bWarningNoBuz : REFERENCE TO BOOL;
	p_bWarning1 : REFERENCE TO BOOL;
	p_bWarning1NoBuz : REFERENCE TO BOOL;
	p_bWarning2 : REFERENCE TO BOOL;
	p_bWarning2NoBuz : REFERENCE TO BOOL;
	p_bWarning3 : REFERENCE TO BOOL;
	p_bWarning3NoBuz : REFERENCE TO BOOL;
	p_bWarning4 : REFERENCE TO BOOL;
	p_bWarning4NoBuz : REFERENCE TO BOOL;
	p_bWarning5 : REFERENCE TO BOOL;
	p_bWarning5NoBuz : REFERENCE TO BOOL;
	p_bChgRcp : REFERENCE TO BOOL;
	p_bSeqStop : REFERENCE TO BOOL;
	p_bStep : REFERENCE TO BOOL;
	p_bOps : REFERENCE TO BOOL;
	p_bStandby : REFERENCE TO BOOL;
	p_bSimulation : REFERENCE TO BOOL;
	p_bMuteBuz : REFERENCE TO BOOL;
END_VAR
(**)
(*TLBuz ChangeRcp Behaviour*)
VAR
	p_tTLChgRcpBlinkTm : REFERENCE TO TIME;
END_VAR
(*TLBuz Error Behaviour*)
VAR
	p_tTLErrBlinkTm : REFERENCE TO TIME;
	p_tBuzErrOnTm : REFERENCE TO TIME;
	p_tBuzErrRestTm : REFERENCE TO TIME;
	p_usiBuzErrOnCntr : REFERENCE TO USINT;
	p_bBuzErrStopSeqEn : REFERENCE TO BOOL;
	p_usiBuzErrStopSeqCntr : REFERENCE TO USINT;
END_VAR
(*TLBuz Default Warning Behaviour*)
VAR
	p_tTLWarnBlinkTm : REFERENCE TO TIME;
	p_tBuzWarnOnTm : REFERENCE TO TIME;
	p_tBuzWarnRestTm : REFERENCE TO TIME;
	p_usiBuzWarnOnCntr : REFERENCE TO USINT;
	p_bBuzWarnStopSeqEn : REFERENCE TO BOOL;
	p_usiBuzWarnStopSeqCntr : REFERENCE TO USINT;
END_VAR
(*TLBuz Special Warning 1 Behaviour*)
VAR
	p_tTLWarn1BlinkTm : REFERENCE TO TIME;
	p_tBuzWarn1OnTm : REFERENCE TO TIME;
	p_tBuzWarn1RestTm : REFERENCE TO TIME;
	p_usiBuzWarn1OnCntr : REFERENCE TO USINT;
	p_bBuzWarn1StopSeqEn : REFERENCE TO BOOL;
	p_usiBuzWarn1StopSeqCntr : REFERENCE TO USINT;
END_VAR
(*TLBuz Special Warning 2 Behaviour*)
VAR
	p_tTLWarn2BlinkTm : REFERENCE TO TIME;
	p_tBuzWarn2OnTm : REFERENCE TO TIME;
	p_tBuzWarn2RestTm : REFERENCE TO TIME;
	p_usiBuzWarn2OnCntr : REFERENCE TO USINT;
	p_bBuzWarn2StopSeqEn : REFERENCE TO BOOL;
	p_usiBuzWarn2StopSeqCntr : REFERENCE TO USINT;
END_VAR
(*TLBuz Special Warning 3 Behaviour*)
VAR
	p_tTLWarn3BlinkTm : REFERENCE TO TIME;
	p_tBuzWarn3OnTm : REFERENCE TO TIME;
	p_tBuzWarn3RestTm : REFERENCE TO TIME;
	p_usiBuzWarn3OnCntr : REFERENCE TO USINT;
	p_bBuzWarn3StopSeqEn : REFERENCE TO BOOL;
	p_usiBuzWarn3StopSeqCntr : REFERENCE TO USINT;
END_VAR
(*TLBuz Special Warning 4 Behaviour*)
VAR
	p_tTLWarn4BlinkTm : REFERENCE TO TIME;
	p_tBuzWarn4OnTm : REFERENCE TO TIME;
	p_tBuzWarn4RestTm : REFERENCE TO TIME;
	p_usiBuzWarn4OnCntr : REFERENCE TO USINT;
	p_bBuzWarn4StopSeqEn : REFERENCE TO BOOL;
	p_usiBuzWarn4StopSeqCntr : REFERENCE TO USINT;
END_VAR
(*TLBuz Special Warning 5 Behaviour*)
VAR
	p_tTLWarn5BlinkTm : REFERENCE TO TIME;
	p_tBuzWarn5OnTm : REFERENCE TO TIME;
	p_tBuzWarn5RestTm : REFERENCE TO TIME;
	p_usiBuzWarn5OnCntr : REFERENCE TO USINT;
	p_bBuzWarn5StopSeqEn : REFERENCE TO BOOL;
	p_usiBuzWarn5StopSeqCntr : REFERENCE TO USINT;
END_VAR
(*TLBuz Special Buz Behaviour*)
VAR
	p_tBuzAlertOnTm : REFERENCE TO TIME;
	p_tBuzAlertRestTm : REFERENCE TO TIME;
	p_usiBuzAlertOnCntr : REFERENCE TO USINT;
	p_bBuzAlertStopSeqEn : REFERENCE TO BOOL;
	p_usiBuzAlertStopSeqCntr : REFERENCE TO USINT;
END_VAR
(*TLBuz Special Ops TL Behaviour*)
VAR
	p_tTLBlueBlinkTm : REFERENCE TO TIME;
	p_tTLAmberBlinkTm : REFERENCE TO TIME;
	p_tTLWhiteBlinkTm : REFERENCE TO TIME;
	p_tTLRedBlinkTm : REFERENCE TO TIME;
	p_tTLGreenBlinkTm : REFERENCE TO TIME;
END_VAR
(**)
VAR
	p_tErrBlinkTm : REFERENCE TO TIME;
	p_tChgRcpBlinkTm : REFERENCE TO TIME;
	p_tWarnBlinkTm : REFERENCE TO TIME;
	p_tWarnRestTm : REFERENCE TO TIME;
	p_usiWarnOnTm : REFERENCE TO USINT;
	p_tWarn1BlinkTm : REFERENCE TO TIME;
	p_tWarn1RestTm : REFERENCE TO TIME;
	p_usiWarn1OnTm : REFERENCE TO USINT;
	p_tWarn2BlinkTm : REFERENCE TO TIME;
	p_tWarn2RestTm : REFERENCE TO TIME;
	p_usiWarn2OnTm : REFERENCE TO USINT;
	p_tWarn3BlinkTm : REFERENCE TO TIME;
	p_tWarn3RestTm : REFERENCE TO TIME;
	p_usiWarn3OnTm : REFERENCE TO USINT;
	p_tWarn4BlinkTm : REFERENCE TO TIME;
	p_tWarn4RestTm : REFERENCE TO TIME;
	p_usiWarn4OnTm : REFERENCE TO USINT;
	p_tWarn5BlinkTm : REFERENCE TO TIME;
	p_tWarn5RestTm : REFERENCE TO TIME;
	p_usiWarn5OnTm : REFERENCE TO USINT;
END_VAR
(**)
VAR
	p_bCoverSwitchSig : REFERENCE TO BOOL;
	p_eTLBuzMode : REFERENCE TO eTLBuzMod;
END_VAR
(**)
VAR
	p_bAOIErrSig : REFERENCE TO BOOL;
	p_bAOIOriginSig : REFERENCE TO BOOL;
	p_bBuzAlertEn : REFERENCE TO BOOL;
	p_bTLBlueFlashEn : REFERENCE TO BOOL;
	p_bTLAmberFlashEn : REFERENCE TO BOOL;
	p_bTLWhiteFlashEn : REFERENCE TO BOOL;
	p_bTLRedFlashEn : REFERENCE TO BOOL;
	p_bTLGreenFlashEn : REFERENCE TO BOOL;
END_VAR
```

#### Local.var - Do Not Change!!!
```iecst
(*2020-10-05*)
(**)
(*Local Action, State & Status*)
VAR
	eAct : eTLBuzAction := TLBuzActIdle;
	eStat : eTLBuzAction := TLBuzActIdle;
	eStatus : eFBStatus := Idle;
	sStatTxt : STRING[200] := '';
	a_sStatText : ARRAY[0..50] OF STRING[200] := ['Idling','Turning On Tower Light Green','Turning On Tower Light Amber','Turning On Tower Light Red','Turning On Buzzer','Turning Off Tower Light Green','Turning Off Tower Light Amber','Turning Off Tower Light Red','Turning Off Buzzer','Turning On All Output','Turning Off All Output',40('')];
END_VAR
(**)
(*Local Alarm*)
(**)
(*Local Output*)
VAR
	bTLRed : BOOL;
	bTLAmber : BOOL;
	bTLGreen : BOOL;
	bTLBlue : BOOL;
	bTLWhite : BOOL;
	bBuzBeep : BOOL;
END_VAR
(**)
(*Local Input*)
VAR
	bManualErrOn : BOOL := FALSE;
	bManual : BOOL := FALSE;
	bStartup : BOOL := FALSE;
	bErr : BOOL := FALSE;
	bErrNoBuz : BOOL := FALSE;
	bWarning : BOOL := FALSE;
	bWarningNoBuz : BOOL := FALSE;
	bWarning1 : BOOL := FALSE;
	bWarning1NoBuz : BOOL := FALSE;
	bWarning2 : BOOL := FALSE;
	bWarning2NoBuz : BOOL := FALSE;
	bWarning3 : BOOL := FALSE;
	bWarning3NoBuz : BOOL := FALSE;
	bWarning4 : BOOL := FALSE;
	bWarning4NoBuz : BOOL := FALSE;
	bWarning5 : BOOL := FALSE;
	bWarning5NoBuz : BOOL := FALSE;
	bChgRcp : BOOL := FALSE;
	bSeqStop : BOOL := FALSE;
	bStep : BOOL := FALSE;
	bOps : BOOL := FALSE;
	bStandby : BOOL := FALSE;
	bSimulation : BOOL := FALSE;
	bMuteBuz : BOOL := FALSE;
END_VAR
(**)
VAR
	tTLChgRcpBlinkTm : TIME := T#200ms;
	tTLErrBlinkTm : TIME := T#500ms;
	tBuzErrOnTm : TIME := T#500ms;
	tBuzErrRestTm : TIME := T#500ms;
	usiBuzErrOnCntr : USINT := 3;
	bBuzErrStopSeqEn : BOOL := FALSE;
	usiBuzErrStopSeqCntr : USINT := 3;
	tTLWarnBlinkTm : TIME := T#500ms;
	tBuzWarnOnTm : TIME := T#500ms;
	tBuzWarnRestTm : TIME := T#5s;
	usiBuzWarnOnCntr : USINT := 3;
	bBuzWarnStopSeqEn : BOOL := FALSE;
	usiBuzWarnStopSeqCntr : USINT := 3;
	tTLWarn1BlinkTm : TIME := T#500ms;
	tBuzWarn1OnTm : TIME := T#500ms;
	tBuzWarn1RestTm : TIME := T#5s;
	usiBuzWarn1OnCntr : USINT := 3;
	bBuzWarn1StopSeqEn : BOOL := FALSE;
	usiBuzWarn1StopSeqCntr : USINT := 3;
	tTLWarn2BlinkTm : TIME := T#500ms;
	tBuzWarn2OnTm : TIME := T#500ms;
	tBuzWarn2RestTm : TIME := T#5s;
	usiBuzWarn2OnCntr : USINT := 3;
	bBuzWarn2StopSeqEn : BOOL := FALSE;
	usiBuzWarn2StopSeqCntr : USINT := 3;
	tTLWarn3BlinkTm : TIME := T#500ms;
	tBuzWarn3OnTm : TIME := T#500ms;
	tBuzWarn3RestTm : TIME := T#5s;
	usiBuzWarn3OnCntr : USINT := 3;
	bBuzWarn3StopSeqEn : BOOL := FALSE;
	usiBuzWarn3StopSeqCntr : USINT := 3;
	tTLWarn4BlinkTm : TIME := T#500ms;
	tBuzWarn4OnTm : TIME := T#500ms;
	tBuzWarn4RestTm : TIME := T#5s;
	usiBuzWarn4OnCntr : USINT := 3;
	bBuzWarn4StopSeqEn : BOOL := FALSE;
	usiBuzWarn4StopSeqCntr : USINT := 3;
	tTLWarn5BlinkTm : TIME := T#500ms;
	tBuzWarn5OnTm : TIME := T#500ms;
	tBuzWarn5RestTm : TIME := T#5s;
	usiBuzWarn5OnCntr : USINT := 3;
	bBuzWarn5StopSeqEn : BOOL := FALSE;
	usiBuzWarn5StopSeqCntr : USINT := 3;
	tBuzAlertOnTm : TIME := T#500ms;
	tBuzAlertRestTm : TIME := T#5s;
	usiBuzAlertOnCntr : USINT := 3;
	bBuzAlertStopSeqEn : BOOL := FALSE;
	usiBuzAlertStopSeqCntr : USINT := 3;
	tTLBlueBlinkTm : TIME := T#500ms;
	tTLAmberBlinkTm : TIME := T#500ms;
	tTLWhiteBlinkTm : TIME := T#500ms;
	tTLRedBlinkTm : TIME := T#500ms;
	tTLGreenBlinkTm : TIME := T#500ms;
END_VAR
(**)
VAR
	tErrBlinkTm : TIME := T#500ms;
	tChgRcpBlinkTm : TIME := T#200ms;
	tWarnBlinkTm : TIME := T#500ms;
	tWarnRestTm : TIME := T#5s;
	usiWarnOnTm : USINT := 3;
	tWarn1BlinkTm : TIME := T#500ms;
	tWarn1RestTm : TIME := T#5s;
	usiWarn1OnTm : USINT := 3;
	tWarn2BlinkTm : TIME := T#500ms;
	tWarn2RestTm : TIME := T#5s;
	usiWarn2OnTm : USINT := 3;
	tWarn3BlinkTm : TIME := T#500ms;
	tWarn3RestTm : TIME := T#5s;
	usiWarn3OnTm : USINT := 3;
	tWarn4BlinkTm : TIME := T#500ms;
	tWarn4RestTm : TIME := T#5s;
	usiWarn4OnTm : USINT := 3;
	tWarn5BlinkTm : TIME := T#500ms;
	tWarn5RestTm : TIME := T#5s;
	usiWarn5OnTm : USINT := 3;
	bCoveSwitchSig : BOOL := FALSE;
	eTLBuzMode : eTLBuzMod := TLBuzModNutek;
END_VAR
(**)
VAR
	bAOIErrSig : BOOL := FALSE;
	bAOIOriginSig : BOOL := FALSE;
	bBuzAlertEn : BOOL := FALSE;
	bTLBlueFlashEn : BOOL := FALSE;
	bTLAmberFlashEn : BOOL := FALSE;
	bTLWhiteFlashEn : BOOL := FALSE;
	bTLRedFlashEn : BOOL := FALSE;
	bTLGreenFlashEn : BOOL := FALSE;
END_VAR
(**)
(*Local*)
VAR
	bInitDone : BOOL;
	bInitialDone : BOOL;
	tBlinkTm : TIME := T#500ms;
	fbBlink : fbTLBuzBlink;
	fbWarning : fbTLBuzWarn;
	eStatOld : eTLBuzAction := TLBuzActIdle;
	usiWarnInfoStateOld : USINT; (*Default buzzer behavior*)
	usiWarnInfoStateNew : USINT; (*Default buzzer behavior*)
	fbBlink1 : fbTLBuzBlink;
	fbBlink2 : fbTLBuzBlink;
	fbBlink3 : fbTLBuzBlink;
	fbBlink4 : fbTLBuzBlink;
	fbWarning1 : fbTLBuzWarn;
END_VAR
```

### Alarm.typ - Do Not Change!!!
```iecst
(*2019-03-25*)
(**)

TYPE
	eAlarmAction :
		(
		AlarmActIdle,
		AlarmActCreateDir,
		AlarmActDeleteOldLog,
		AlarmActReadHistory,
		AlarmActWriteHistory,
		AlarmActAppendLog,
		AlarmActAppendLogWriteHistory,
		AlarmActResetHistory,
		AlarmActBGStartLog,
		AlarmActBGStopLog
		);
END_TYPE

(**)

TYPE
	tyAlarmCurr : 	STRUCT
		eSeverity : eAlmSeverity;
		sMsg : STRING[300];
		bAlm : BOOL;
		bWarning : BOOL;
		udiErrorCode : UDINT;
		sProgNm : STRING[15];
		sDT : STRING[80];
		udiModErrCode : UDINT;
	END_STRUCT;
	tyHistory : 	STRUCT
		sDT : STRING[80];
		sProgNm : STRING[15];
		udiModErrCode : UDINT;
		udiErrorCode : UDINT;
	END_STRUCT;
END_TYPE
```

### Alarm.var - Change By Project
```iecst
(*2019-03-25*)
(**)
(*Constant*)
VAR CONSTANT
	c_udiAlarmCurrMax : UDINT := 200;
	c_udiAlarmHistoryMax : UDINT := 300;
	c_udiAlarmMaxModule : UDINT := 60;
	c_udiAlarminfoMaxModule : UDINT := 10;
END_VAR
(**)
(*Action & State & Status*)
VAR
	p_AlarmStat : UDINT;
	p_AlarmStatus : UDINT;
	p_AlarmStatTxt : UDINT;
END_VAR
(**)
(*Alarm*)
(**)
(*Output*)
VAR
	p_AlarmErr : UDINT;
	p_AlarmWarning : UDINT;
	p_AlarmCurrList : UDINT;
	p_AlarmRecoveryList : UDINT;
	p_AlarmHistoryList : UDINT;
	p_AlarmInfo : UDINT;
	p_AlarmInfoLF : UDINT;
	p_AlarmInfoMsg : UDINT;
	p_AlarmHistoryFileNotFound : UDINT;
END_VAR
(**)
(**)
(*Alarm Program Name: Declare Global Variables Based on the Projects' Packages.*)
VAR
	g_sAWOpenProgNm : STRING[15];
	g_sAWCloseProgNm : STRING[15];
	g_sMagAWOpenProgNm : STRING[15];
	g_sTravProgNm : STRING[15];
	g_sLifterBtmProgNm : STRING[15];
	g_sConvProgNm : STRING[15];
	g_sDCConvProgNm : STRING[15];
	g_sMagConvProgNm : STRING[15];
	g_sMagConv2ClpProgNm : STRING[15];
	g_sBufferProgNm : STRING[15];
	g_sMotorBrkProgNm : STRING[15];
	g_sMtrPshrProgNm : STRING[15];
	g_sStepperProgNm : STRING[15];
	g_sPneuNoSenProgNm : STRING[15];
	g_sPneuExtSenProgNm : STRING[15];
	g_sPneuRetSenProgNm : STRING[15];
	g_sPneu2SenProgNm : STRING[15];
	g_sPneu3SenProgNm : STRING[15];
	g_sUSSMEMAProgNm : STRING[15];
	g_sDSSMEMAProgNm : STRING[15];
	g_sHermesProgNm : STRING[15];
	g_sUSHermesProgNm : STRING[15];
	g_sDSHermesProgNm : STRING[15];
	g_sRmtHermesProgNm : STRING[15];
	g_sLFLeaderProgNm : STRING[15];
	g_sLFFollowerProgNm : STRING[15];
	g_sLCSProgNm : STRING[15];
	g_sLCSLFProgNm : STRING[15];
	g_sLCSMngRcpProgNm : STRING[15];
	g_sTCPProgNm : STRING[15];
	g_sUSSOTProgNm : STRING[15];
	g_sDSSOTProgNm : STRING[15];
	g_sBarcodeRdrProgNm : STRING[15];
	g_sRS232MirtecProgNm : STRING[15];
	g_sProdRcpProgNm : STRING[15];
	g_sMagRcpProgNm : STRING[15];
	g_sMpProdRcpProgNm : STRING[15];
	g_sAlarmProgNm : STRING[15];
	g_sNtParamProgNm : STRING[15];
	g_sMcParamProgNm : STRING[15];
	g_sUsrMgmtProgNm : STRING[15];
	g_sLibVerProgNm : STRING[15];
	g_sUsrFolderProgNm : STRING[15];
	g_sHWInfoProgNm : STRING[15];
	g_sDInputProgNm : STRING[15];
	g_sTimeProgNm : STRING[15];
	g_sMachineProgNm : STRING[15];
	g_sOpsInvertProgNm : STRING[15];
	g_sLiberWarnName : STRING[15];
	g_sOps2ProgNm : STRING[15];
	g_sOps3ProgNm : STRING[15];
	g_sOps4ProgNm : STRING[15];
END_VAR
(**)
```

### Program Logical/Alarm/Alarm (IEC, version 1.00.0) - 1.00.0 - NtLogFile v5.00.0 , NtFileIO v5.00.0

#### Init.st - Change By Project
```iecst
(** 2021-04-20 **)
PROGRAM _INIT

	(* Always Change If Project Change *)

	//Pass Address To Global Address For External Use
	//Action, State & Status
	p_AlarmStat		:= ADR(eStat);
	p_AlarmStatus	:= ADR(eStatus);
	p_AlarmStatTxt	:= ADR(sStatTxt);

	//Alarm

	//Output
	p_AlarmErr					:= ADR(bErr);
	p_AlarmWarning				:= ADR(bWarning);
	p_AlarmCurrList				:= ADR(a_tyCurrList);
	p_AlarmRecoveryList			:= ADR(a_udiRecoveryList);
	p_AlarmHistoryList			:= ADR(a_sHistoryList);
	p_AlarmInfo					:= ADR(bInfo);
	p_AlarmInfoLF				:= ADR(bInfoLF);
	p_AlarmInfoMsg				:= ADR(sInfoMsg);
	p_AlarmHistoryFileNotFound	:= ADR(bHistoryFileNotFound);

	(* Always Change If Project Change *)

END_PROGRAM
```

#### Act_InitGlobal.st - Change By Project
```iecst
(** 2020-09-10 **)
ACTION Act_InitGlobal:

	(* Always Change If Project Change *)

	//Pass Data To Link
	p_tyLinkDIAlmData1 ACCESS p_DIAlmData1;
	p_tyLinkDIAlmData2 ACCESS p_DIAlmData2;
	p_tyLinkUsrMgmtAlmData ACCESS p_UsrMgmtAlmData;
	p_tyLinkUSSMEMAAlmData ACCESS p_USSMEMAAlmData;
	p_tyLinkDSSMEMAAlmData ACCESS p_DSSMEMAAlmData;
	p_tyLinkUSSMEMA2AlmData ACCESS p_USSMEMA2AlmData;
	p_tyLinkMcParamAlmData ACCESS p_McParamAlmData;
	p_tyLinkNtParamAlmData ACCESS p_NtParamAlmData;
	p_tyLinkProdRcpAlmData ACCESS p_ProdRcpAlmData;
	p_tyLinkAWAlmData ACCESS p_AWOpenAlmData;
	p_tyLinkAWAlmData1 ACCESS p_AWOpenAlmData1;
	p_tyLinkAWAlmData2 ACCESS p_AWOpenAlmData2;
	p_tyLinkAWAlmData3 ACCESS p_AWOpenAlmData3;
	p_tyLinkMotorBrkAlmData ACCESS p_MotorBrkAlmData;
	p_tyLinkTimeAlmData	ACCESS p_TimeAlmData;
	p_tyLinkTimeAlmData1 ACCESS p_TimeAlmData1;
	p_tyLinkUsrFolderAlmData ACCESS p_UsrFolderAlmData;
	p_tyLinkLibVerAlmData ACCESS p_LibVerAlmData;
	p_tyLinkHWInfoAlmData ACCESS p_HWInfoAlmData;
	p_tyLinkConvAlmData ACCESS p_ConvAlmData;
	p_tyLinkMcAlmData ACCESS p_McAlmData;
	p_tyLinkMcAlmData1 ACCESS p_McAlmData1;
	p_tyLinkPneuNoSenStopperAlmData ACCESS p_PneuNoSenStopperAlmData;
	p_tyLinkPneuNoSenClampAlmData ACCESS p_PneuNoSenClampAlmData;
	p_tyLinkOpsInvertAlmData ACCESS p_OpsInvertAlmData;
	p_tyLinkOpsInvertAlmData1 ACCESS p_OpsInvertAlmData1;
	p_tyLinkHermesAlmData ACCESS p_HermesAlmData;
	p_tyLinkUSHermesAlmData ACCESS p_USHermesAlmData;
	p_tyLinkUSHermesAlmData1 ACCESS p_USHermesAlmData1;
	p_tyLinkUSHermesAlmData2 ACCESS p_USHermesAlmData2;
	p_tyLinkUSHermesAlmData3 ACCESS p_USHermesAlmData3;
	p_tyLinkUSHermesAlmData4 ACCESS p_USHermesAlmData4;
	p_tyLinkUSHermesAlmData5 ACCESS p_USHermesAlmData5;
	p_tyLinkUSHermesInfoData ACCESS p_USHermesInfoData;
	p_tyLinkDSHermesAlmData ACCESS p_DSHermesAlmData;
	p_tyLinkDSHermesAlmData1 ACCESS p_DSHermesAlmData1;
	p_tyLinkDSHermesAlmData2 ACCESS p_DSHermesAlmData2;
	p_tyLinkDSHermesAlmData3 ACCESS p_DSHermesAlmData3;
	p_tyLinkDSHermesAlmData4 ACCESS p_DSHermesAlmData4;
	p_tyLinkDSHermesInfoData ACCESS p_DSHermesInfoData;
	p_tyLinkLFLeaderAlmData ACCESS p_LFLeaderAlmData;
	p_tyLinkLFFollowerAlmData ACCESS p_LFFollowerAlmData;
	p_tyLinkLFFollowerInfoData ACCESS p_LFFollowerInfoData;
	p_tyLinkLFFollowerInfoData1 ACCESS p_LFFollowerInfoData1;
	p_tyLinkFollower1AlmData ACCESS p_Follower1AlmData;
	p_tyLinkFollower1InfoData ACCESS p_Follower1InfoData;
	p_tyLinkFollower1InfoData1 ACCESS p_Follower1InfoData1;
	p_tyLinkLCSMngRcpAlmData ACCESS p_LCSMngRcpAlmData;
	p_tyLinkLCSLFAlmData ACCESS p_LCSLFAlmData;
	p_tyLinkLCSLFInfoData ACCESS p_LCSLFInfoData;
	p_tyLinkMpProdRcpAlmData ACCESS p_MpProdRcpAlmData;
	p_tyLinkPneu2SenInShutterAlmData ACCESS p_Pneu2SenInShutterAlmData;
	p_tyLinkPneu2SenOutShuttrAlmData ACCESS p_Pneu2SenOutShutterAlmData;
	p_tyLinkPneu2SenClamp1AlmData ACCESS p_Pneu2SenClamp1AlmData;
	p_tyLinkPneu2SenClamp2AlmData ACCESS p_Pneu2SenClamp2AlmData;
	p_tyLinkPneu2SenClamp3AlmData ACCESS p_Pneu2SenClamp3AlmData;

	//Pass Data To Internal Use
	p_udiRstErr ACCESS p_RstErrReset;
	p_eAct ACCESS p_StartupAlarmAct;
	p_dtCurrDT ACCESS p_TimeCurrDT;
	p_udiFileKeepDay ACCESS p_NtParamAlmFileKeepDay;
	p_sProgNm ACCESS p_NtParamAlmProgNm;
	p_bNtSettingsLoadDone ACCESS p_StartupNtSettingsLoadDone;
	p_bStartupUISettingsLoadDone ACCESS p_StartupUISettingsLoadDone;

	(* Always Change If Project Change *)

END_ACTION
```

#### InputRef_Link.var - Change By Project
```iecst
(*2019-01-07*)
(**)
(*External Data*)
VAR
	p_tyLinkDIAlmData1 : REFERENCE TO tyAlmDat;
	p_tyLinkDIAlmData2 : REFERENCE TO tyAlmDat;
	p_tyLinkUsrMgmtAlmData : REFERENCE TO tyAlmDat;
	p_tyLinkUSSMEMAAlmData : REFERENCE TO tyAlmDat;
	p_tyLinkDSSMEMAAlmData : REFERENCE TO tyAlmDat;
	p_tyLinkUSSMEMA2AlmData : REFERENCE TO tyAlmDat;
	p_tyLinkMcParamAlmData : REFERENCE TO tyAlmDat;
	p_tyLinkNtParamAlmData : REFERENCE TO tyAlmDat;
	p_tyLinkProdRcpAlmData : REFERENCE TO tyAlmDat;
	p_tyLinkAWAlmData : REFERENCE TO tyAlmDat;
	p_tyLinkAWAlmData1 : REFERENCE TO tyAlmDat;
	p_tyLinkAWAlmData2 : REFERENCE TO tyAlmDat;
	p_tyLinkAWAlmData3 : REFERENCE TO tyAlmDat;
	p_tyLinkMotorBrkAlmData : REFERENCE TO tyAlmDat;
	p_tyLinkTimeAlmData : REFERENCE TO tyAlmDat;
	p_tyLinkTimeAlmData1 : REFERENCE TO tyAlmDat;
	p_tyLinkUsrFolderAlmData : REFERENCE TO tyAlmDat;
	p_tyLinkLibVerAlmData : REFERENCE TO tyAlmDat;
	p_tyLinkHWInfoAlmData : REFERENCE TO tyAlmDat;
	p_tyLinkConvAlmData : REFERENCE TO tyAlmDat;
	p_tyLinkMcAlmData : REFERENCE TO tyAlmDat;
	p_tyLinkMcAlmData1 : REFERENCE TO tyAlmDat;
	p_tyLinkPneuNoSenStopperAlmData : REFERENCE TO tyAlmDat;
	p_tyLinkPneuNoSenClampAlmData : REFERENCE TO tyAlmDat;
	p_tyLinkPneu2SenInShutterAlmData : REFERENCE TO tyAlmDat;
	p_tyLinkPneu2SenOutShuttrAlmData : REFERENCE TO tyAlmDat;
	p_tyLinkPneu2SenClamp1AlmData : REFERENCE TO tyAlmDat;
	p_tyLinkPneu2SenClamp2AlmData : REFERENCE TO tyAlmDat;
	p_tyLinkPneu2SenClamp3AlmData : REFERENCE TO tyAlmDat;
	p_tyLinkOpsInvertAlmData : REFERENCE TO tyAlmDat;
	p_tyLinkOpsInvertAlmData1 : REFERENCE TO tyAlmDat;
	p_tyLinkHermesAlmData : REFERENCE TO tyAlmDat;
	p_tyLinkUSHermesAlmData : REFERENCE TO tyAlmDat;
	p_tyLinkUSHermesAlmData1 : REFERENCE TO tyAlmDat;
	p_tyLinkUSHermesAlmData2 : REFERENCE TO tyAlmDat;
	p_tyLinkUSHermesAlmData3 : REFERENCE TO tyAlmDat;
	p_tyLinkUSHermesAlmData4 : REFERENCE TO tyAlmDat;
	p_tyLinkUSHermesAlmData5 : REFERENCE TO tyAlmDat;
	p_tyLinkUSHermesInfoData : REFERENCE TO tyAlmDat;
	p_tyLinkDSHermesAlmData : REFERENCE TO tyAlmDat;
	p_tyLinkDSHermesAlmData1 : REFERENCE TO tyAlmDat;
	p_tyLinkDSHermesAlmData2 : REFERENCE TO tyAlmDat;
	p_tyLinkDSHermesAlmData3 : REFERENCE TO tyAlmDat;
	p_tyLinkDSHermesAlmData4 : REFERENCE TO tyAlmDat;
	p_tyLinkDSHermesInfoData : REFERENCE TO tyAlmDat;
	p_tyLinkLFLeaderAlmData : REFERENCE TO tyAlmDat;
	p_tyLinkLFFollowerAlmData : REFERENCE TO tyAlmDat;
	p_tyLinkLFFollowerInfoData : REFERENCE TO tyAlmDat;
	p_tyLinkLFFollowerInfoData1 : REFERENCE TO tyAlmDat;
	p_tyLinkFollower1AlmData : REFERENCE TO tyAlmDat;
	p_tyLinkFollower1InfoData : REFERENCE TO tyAlmDat;
	p_tyLinkFollower1InfoData1 : REFERENCE TO tyAlmDat;
	p_tyLinkLCSMngRcpAlmData : REFERENCE TO tyAlmDat;
	p_tyLinkLCSLFAlmData : REFERENCE TO tyAlmDat;
	p_tyLinkLCSLFInfoData : REFERENCE TO tyAlmDat;
	p_tyLinkMpProdRcpAlmData : REFERENCE TO tyAlmDat;
END_VAR
(**)
VAR
	fbDlyTmr : TON := (PT:=T#5s);
	fbDeleteLogTmr : TON := (PT:=T#24h);
END_VAR
(**)
```

#### Act_LinkAction.st - Change By Project
```iecst
(** 2019-03-29 **)
ACTION Act_LinkAction:

	//Delete Old Alarm Log File for 24 hours After Machine is Continuous Running 30 Days.

	fbDlyTmr(IN := TRUE);
	IF fbDlyTmr.Q THEN
		fbDeleteLogTmr (IN := TRUE);
		IF fbDeleteLogTmr.Q AND eStatus <> Busy THEN
			p_eAct := AlarmActDeleteOldLog;
			IF eStat = AlarmActDeleteOldLog AND eStatus = Done THEN
				p_eAct := AlarmActIdle;
				fbDlyTmr (IN := FALSE);
				fbDeleteLogTmr (IN := FALSE);
			END_IF
		END_IF
	END_IF

END_ACTION
```

#### Act_Link.st - Change By Project
```iecst
(** 2020-09-10 **)
ACTION Act_Link:

	//Index 1 For Internal Use
	pa_tyAlmData[2]		:= p_tyLinkDIAlmData1;
	pa_tyAlmData[3]		:= p_tyLinkDIAlmData2;
	pa_tyAlmData[4]		:= p_tyLinkUsrMgmtAlmData;
	pa_tyAlmData[5]		:= p_tyLinkUSSMEMAAlmData;
	pa_tyAlmData[6]		:= p_tyLinkDSSMEMAAlmData;
	pa_tyAlmData[7]		:= p_tyLinkMcParamAlmData;
	pa_tyAlmData[8]		:= p_tyLinkNtParamAlmData;
	pa_tyAlmData[9]		:= p_tyLinkProdRcpAlmData;
	pa_tyAlmData[10]	:= p_tyLinkAWAlmData;
	pa_tyAlmData[11]	:= p_tyLinkAWAlmData1;
	pa_tyAlmData[12]	:= p_tyLinkAWAlmData2;
	pa_tyAlmData[13]	:= p_tyLinkAWAlmData3;
	pa_tyAlmData[18]	:= p_tyLinkTimeAlmData;
	pa_tyAlmData[19]	:= p_tyLinkTimeAlmData1;
	pa_tyAlmData[20]	:= p_tyLinkUsrFolderAlmData;
	pa_tyAlmData[21]	:= p_tyLinkLibVerAlmData;
	pa_tyAlmData[22]	:= p_tyLinkHWInfoAlmData;
	pa_tyAlmData[23]	:= p_tyLinkConvAlmData;
	pa_tyAlmData[24]	:= p_tyLinkMcAlmData;
	pa_tyAlmData[25]	:= p_tyLinkMcAlmData1;
	pa_tyAlmData[26]	:= p_tyLinkPneuNoSenStopperAlmData;
	pa_tyAlmData[28]	:= p_tyLinkOpsInvertAlmData;
	pa_tyAlmData[29]	:= p_tyLinkHermesAlmData;
	pa_tyAlmData[30]	:= p_tyLinkUSHermesAlmData;
	pa_tyAlmData[31]	:= p_tyLinkUSHermesAlmData1;
	pa_tyAlmData[32]	:= p_tyLinkUSHermesAlmData2;
	pa_tyAlmData[33]	:= p_tyLinkUSHermesAlmData3;
	pa_tyAlmData[34]	:= p_tyLinkUSHermesAlmData4;
	pa_tyAlmData[35]	:= p_tyLinkUSHermesAlmData5;
	pa_tyAlmData[36]	:= p_tyLinkUSHermesInfoData;
	pa_tyAlmData[37]	:= p_tyLinkDSHermesAlmData;
	pa_tyAlmData[38]	:= p_tyLinkDSHermesAlmData1;
	pa_tyAlmData[39]	:= p_tyLinkDSHermesAlmData2;
	pa_tyAlmData[40]	:= p_tyLinkDSHermesAlmData3;
	pa_tyAlmData[41]	:= p_tyLinkDSHermesAlmData4;
	pa_tyAlmData[42]	:= p_tyLinkLFLeaderAlmData;
	pa_tyAlmData[43]	:= p_tyLinkLFFollowerAlmData;
	pa_tyAlmData[44]	:= p_tyLinkLFFollowerInfoData;
	pa_tyAlmData[45]	:= p_tyLinkLFFollowerInfoData1;
	pa_tyAlmData[46]	:= p_tyLinkFollower1AlmData;
	pa_tyAlmData[47]	:= p_tyLinkFollower1InfoData;
	pa_tyAlmData[48]	:= p_tyLinkFollower1InfoData1;
	pa_tyAlmData[49]	:= p_tyLinkLCSMngRcpAlmData;
	pa_tyAlmData[50]	:= p_tyLinkLCSLFAlmData;
	pa_tyAlmData[51]	:= p_tyLinkLCSLFInfoData;
	pa_tyAlmData[52]	:= p_tyLinkMpProdRcpAlmData;
	pa_tyAlmData[53]	:= p_tyLinkMotorBrkAlmData;
	pa_tyAlmData[54]	:= p_tyLinkPneuNoSenClampAlmData;
	pa_tyAlmData[55]	:= p_tyLinkPneu2SenInShutterAlmData;
	pa_tyAlmData[56]	:= p_tyLinkPneu2SenOutShuttrAlmData;
	pa_tyAlmData[57]	:= p_tyLinkPneu2SenClamp1AlmData;
	pa_tyAlmData[58]	:= p_tyLinkPneu2SenClamp2AlmData;
	pa_tyAlmData[59]	:= p_tyLinkPneu2SenClamp3AlmData;
	pa_tyAlmData[60]	:= p_tyLinkUSSMEMA2AlmData;
	pa_tyAlmData[61]	:= p_tyLinkOpsInvertAlmData1;
	pa_tyAlmData[62]	:= p_tyLinkDSHermesInfoData;
END_ACTION
```

#### Cyclic.st - Do Not Change!!!
```iecst
(** 2019-03-29 **)
PROGRAM _CYCLIC

	IF bInitDone = FALSE THEN
		bInitDone	:= TRUE;

		Act_InitLocal;
		Act_InitGlobal;

	ELSIF bInitialDone = FALSE THEN
		IF p_bNtSettingsLoadDone = TRUE THEN
			bInitialDone	:= TRUE;

			Act_Initial;
		END_IF

	ELSE

		Act_Background;
		Act_RstErr;
		Act_LinkAction;
		Act_Action;
		Act_Link;
		Act_Main;
		Act_Alarm;

	END_IF

END_PROGRAM
```

#### Act_RstErr.st - Do Not Change!!!
```iecst
(** 2020-07-27 **)
ACTION Act_RstErr:

	IF p_udiRstErr <> udiRstErrOld THEN
		bRstErr			:= TRUE;
		udiRstErrOld	:= p_udiRstErr;
	ELSE
		bRstErr			:= FALSE;
	END_IF

	//Checking which Warning is clear
	IF a_tyWarningCurrList[1].sMsg <> '' AND p_tyLinkLibVerAlmData.udiCode = 0 THEN

		FOR udi2 := 1 TO (udiWarningMax-1) DO
			udiRecorded1:= udiRecorded[udi2];
			IF 	(pa_tyAlmData[udiRecorded1].eSeverity =  AlmSeverityNA) AND udiRecorded1<> 0 THEN
				bRstWarning := TRUE;
				EXIT;
			ELSE
				bRstWarning := FALSE;
			END_IF

		END_FOR
	ELSE
		bRstWarning := FALSE;
	END_IF

END_ACTION
```

#### Act_InitLocal.st - Do Not Change!!!
```iecst
(** 2019-03-25 **)
ACTION Act_InitLocal:

	//Input Reference Link To Local Variable
	p_eAct ACCESS ADR(eAct);
	p_udiCurrMax ACCESS ADR(c_udiAlarmCurrMax);
	p_udiHistoryMax ACCESS ADR(c_udiAlarmHistoryMax);
	p_udiRstErr ACCESS ADR(udiRstErr);
	p_dtCurrDT ACCESS ADR(dtCurrDT);
	pa_tyAlmData ACCESS ADR(a_tyAlmData);
	p_udiFileKeepDay ACCESS ADR(udiFileKeepDay);
	p_sProgNm ACCESS ADR(sProgNm);
	p_bNtSettingsLoadDone ACCESS ADR(bNtSettingsLoadDone);

END_ACTION
```

#### Act_Initial.st - Do Not Change!!!
```iecst
(** 2019-01-03 **)
ACTION Act_Initial:

	//Initial
	sStatTxt	:= a_sStatText[eStat];

	fbDirCreate1.sDevice	:= 'F';
	fbDirCreate1.sDirName	:= 'User';
	fbDirCreate1(bEn := FALSE);

	fbDirCreate2.sDevice	:= 'User';
	fbDirCreate2.sDirName	:= 'Alarm';
	fbDirCreate2(bEn := FALSE);

	fbFileAppend1.sDevice	:= 'Alarm';
	fbFileAppend1(bEn := FALSE);

	fbFileOldDel1.sDevice	:= 'Alarm';
	fbFileOldDel1.sPath		:= '';
	fbFileOldDel1.sKeyword	:= 'ALARM_';
	fbFileOldDel1(bEn := FALSE);

	fbFileRead1.sDevice		:= 'Alarm';
	fbFileRead1.sFile		:= 'History.dat';
	fbFileRead1.udiOffset	:= 0;
	fbFileRead1.p_Dest		:= ADR(a_tyHistoryList);
	fbFileRead1.udiLen		:= SIZEOF(a_tyHistoryList);
	fbFileRead1(bEn := FALSE);

	fbFileWrite1.sDevice	:= 'Alarm';
	fbFileWrite1.sFile		:= 'History.dat';
	fbFileWrite1.udiOffset	:= 0;
	fbFileWrite1.p_Src		:= ADR(a_tyHistoryList);
	fbFileWrite1.udiLen		:= SIZEOF(a_tyHistoryList);
	fbFileWrite1.udiOption	:= 0;
	fbFileWrite1(bEn := FALSE);

END_ACTION
```

#### Act_Action.st - Do Not Change!!!
```iecst
(** 2019-03-25 **)
ACTION Act_Action:

	//Reset Error
	IF (eStatus = Error) AND bRstErr THEN
		p_eAct	:= AlarmActIdle;
		eStat	:= AlarmActIdle;
	END_IF

	//Reset Done
	IF eStatus = Done AND p_eAct = AlarmActIdle THEN
		eStat	:= AlarmActIdle;
	END_IF

	//Set p_eAct
	IF eStatus = Idle THEN
		eStat	:= p_eAct;
	END_IF

END_ACTION
```

#### Act_Main.st - Do Not Change!!!
```iecst
(** 2019-02-23 **)
ACTION Act_Main:

	//Main
	CASE eStat OF

		AlarmActIdle:
			IF eStatus <> Idle THEN	//Reset Data
				//Private
				fbDirCreate1(bEn := FALSE);
				fbDirCreate2(bEn := FALSE);
				fbFileOldDel1(bEn := FALSE);
				fbFileRead1(bEn := FALSE);
				fbFileAppend1(bEn := FALSE);
				fbFileWrite1(bEn := FALSE);
				usiStep	:= 0;

				bHistoryFileNotFound	:= FALSE;
				udiWriteLogCntr			:= 1;

				sStatTxt	:= a_sStatText[eStat];

			END_IF

			eStatus	:= Idle;

		AlarmActCreateDir:
			IF eStatus = Idle OR eStatus = Busy THEN

				eStatus	:= Busy;

				sStatTxt	:= a_sStatText[eStat];

				CASE usiStep OF
					0:
						fbDirCreate1(bEn := TRUE);
						IF fbDirCreate1.udiStatus = 0 THEN
							usiStep	:= 1;
						ELSIF fbDirCreate1.udiStatus < 65534 THEN
							eStatus		:= Error;

							IF fbDirCreate1.udiStatus = 1908 THEN
								udiStatus	:= 10000;	//Create User Directory Error
							ELSE
								udiStatus	:= fbDirCreate1.udiStatus;
							END_IF
						END_IF

					1:
						fbDirCreate2(bEn := TRUE);
						IF fbDirCreate2.udiStatus = 0 THEN
							eStatus	:= Done;
						ELSIF fbDirCreate2.udiStatus < 65534 THEN
							eStatus		:= Error;

							IF fbDirCreate2.udiStatus = 1908 THEN
								udiStatus	:= 10001;	//Create Alarm Directory Error
							ELSE
								udiStatus	:= fbDirCreate2.udiStatus;
							END_IF
						END_IF

				END_CASE

			END_IF

		AlarmActDeleteOldLog:
			IF eStatus = Idle OR eStatus = Busy THEN

				eStatus	:= Busy;

				sStatTxt	:= a_sStatText[eStat];

				fbFileOldDel1.dtDTNow			:= p_dtCurrDT;
				fbFileOldDel1.udiFileKeepDay	:= p_udiFileKeepDay;
				fbFileOldDel1(bEn := TRUE);
				IF fbFileOldDel1.udiStatus = 0 THEN
					eStatus	:= Done;
				ELSIF fbFileOldDel1.udiStatus < 65534 THEN
					eStatus		:= Error;

					IF fbFileOldDel1.udiStatus = 1910 THEN
						udiStatus	:= 10002;	//Get Directory Info Error While Deleting Old Log
					ELSIF fbFileOldDel1.udiStatus = 1911 THEN
						udiStatus	:= 10003;	//Directory Read Error While Deleting Old Log
					ELSIF fbFileOldDel1.udiStatus = 1912 THEN
						udiStatus	:= 10004;	//File Delete Error While Deleting Old Log
					ELSE
						udiStatus	:= fbFileOldDel1.udiStatus;
					END_IF
				END_IF

			END_IF

		AlarmActReadHistory:
			IF eStatus = Idle OR eStatus = Busy THEN

				eStatus	:= Busy;

				sStatTxt	:= a_sStatText[eStat];

				fbFileRead1(bEn := TRUE);
				IF fbFileRead1.udiStatus = 0 THEN
					eStatus	:= Done;
				ELSIF fbFileRead1.udiStatus < 65534 THEN
					eStatus		:= Error;

					IF fbFileRead1.udiStatus = 1900 THEN
						udiStatus	:= 10005;	//File Open Error While Reading Alarm History
					ELSIF fbFileRead1.udiStatus = 1902 THEN
						udiStatus	:= 10006;	//File Read Error While Reading Alarm History
					ELSIF fbFileRead1.udiStatus = 1904 THEN
						udiStatus	:= 10007;	//File Close Error While Reading Alarm History
					ELSIF fbFileRead1.udiStatus = 1915 THEN
						eStatus					:= Done;
						bHistoryFileNotFound	:= TRUE;
					ELSE
						udiStatus	:= fbFileRead1.udiStatus;
					END_IF
				END_IF

			END_IF

		AlarmActWriteHistory:
			IF eStatus = Idle OR eStatus = Busy THEN

				eStatus	:= Busy;

				sStatTxt	:= a_sStatText[eStat];

				fbFileWrite1(bEn := TRUE);
				IF fbFileWrite1.udiStatus = 0 THEN
					eStatus	:= Done;
				ELSIF fbFileWrite1.udiStatus < 65534 THEN
					eStatus		:= Error;

					IF fbFileWrite1.udiStatus = 1900 THEN
						udiStatus	:= 10008;	//File Open Error While Writing Alarm History
					ELSIF fbFileWrite1.udiStatus = 1901 THEN
						udiStatus	:= 10009;	//File Create Error While Writing Alarm History
					ELSIF fbFileWrite1.udiStatus = 1903 THEN
						udiStatus	:= 10010;	//File Write Error While Writing Alarm History
					ELSIF fbFileWrite1.udiStatus = 1904 THEN
						udiStatus	:= 10011;	//File Close Error While Writing Alarm History
					ELSIF fbFileWrite1.udiStatus = 1914 THEN
						udiStatus	:= 10012;	//Directory Does Not Exist While Writing Alarm History
					ELSE
						udiStatus	:= fbFileWrite1.udiStatus;
					END_IF
				END_IF

			END_IF

		AlarmActAppendLog:
			IF eStatus = Idle OR eStatus = Busy THEN

				eStatus	:= Busy;

				sStatTxt	:= a_sStatText[eStat];

				dtCurrDTTemp			:= p_dtCurrDT;
				fbFileAppend1.sFile		:= DT_TO_STRING(dtCurrDTTemp);
				fbFileAppend1.sFile		:= MID(fbFileAppend1.sFile , 10 , 4);
				fbFileAppend1.sFile		:= CONCAT('ALARM_' , fbFileAppend1.sFile);
				fbFileAppend1.sFile		:= CONCAT(fbFileAppend1.sFile , '.dat');

				fbFileAppend1.p_Src		:= ADR(a_sLogList[udiWriteLogCntr]);
				fbFileAppend1.udiLen	:= LEN(a_sLogList[udiWriteLogCntr]);

				fbFileAppend1(bEn := TRUE);
				IF fbFileAppend1.udiStatus = 0 THEN
					IF udiWriteLogCntr >= udiLogCntr THEN
						eStatus	:= Done;
					ELSE
						udiWriteLogCntr	:= udiWriteLogCntr + 1;
						fbFileAppend1(bEn := FALSE);
					END_IF

				ELSIF fbFileAppend1.udiStatus < 65534 THEN
					eStatus		:= Error;

					IF fbFileAppend1.udiStatus = 1900 THEN
						udiStatus	:= 10013;	//File Open Error While Writing Alarm Log
					ELSIF fbFileAppend1.udiStatus = 1901 THEN
						udiStatus	:= 10014;	//File Create Error While Writing Alarm Log
					ELSIF fbFileAppend1.udiStatus = 1913 THEN
						udiStatus	:= 10015;	//Get File Info Error While Writing Alarm Log
					ELSIF fbFileAppend1.udiStatus = 1903 THEN
						udiStatus	:= 10016;	//File Write Error While Writing Alarm Log
					ELSIF fbFileAppend1.udiStatus = 1904 THEN
						udiStatus	:= 10017;	//File Close Error While Writing Alarm Log
					ELSIF fbFileAppend1.udiStatus = 1914 THEN
						udiStatus	:= 10018;	//Directory Does Not Exist While Writing Alarm Log
					ELSE
						udiStatus	:= fbFileAppend1.udiStatus;
					END_IF
				END_IF

			END_IF

		AlarmActAppendLogWriteHistory:
			IF eStatus = Idle OR eStatus = Busy THEN

				eStatus	:= Busy;

				sStatTxt	:= a_sStatText[eStat];

				dtCurrDTTemp			:= p_dtCurrDT;
				fbFileAppend1.sFile		:= DT_TO_STRING(dtCurrDTTemp);
				fbFileAppend1.sFile		:= MID(fbFileAppend1.sFile , 10 , 4);
				fbFileAppend1.sFile		:= CONCAT('ALARM_' , fbFileAppend1.sFile);
				fbFileAppend1.sFile		:= CONCAT(fbFileAppend1.sFile , '.dat');

				fbFileAppend1.p_Src		:= ADR(a_sLogList[udiWriteLogCntr]);
				fbFileAppend1.udiLen	:= LEN(a_sLogList[udiWriteLogCntr]);

				fbFileAppend1(bEn := TRUE);
				fbFileWrite1(bEn := TRUE);

				IF (fbFileAppend1.udiStatus = 0) AND (udiWriteLogCntr >= udiLogCntr) AND fbFileWrite1.udiStatus = 0 THEN
					eStatus	:= Done;

				ELSIF fbFileAppend1.udiStatus = 0 AND udiWriteLogCntr < udiLogCntr THEN
					udiWriteLogCntr	:= udiWriteLogCntr + 1;
					fbFileAppend1(bEn := FALSE);

				ELSIF fbFileWrite1.udiStatus > 0 AND fbFileWrite1.udiStatus < 65534 THEN
					eStatus		:= Error;

					IF fbFileWrite1.udiStatus = 1900 THEN
						udiStatus	:= 10019;	//File Open Error While Writing Alarm History
					ELSIF fbFileWrite1.udiStatus = 1901 THEN
						udiStatus	:= 10020;	//File Create Error While Writing Alarm History
					ELSIF fbFileWrite1.udiStatus = 1903 THEN
						udiStatus	:= 10021;	//File Write Error While Writing Alarm History
					ELSIF fbFileWrite1.udiStatus = 1904 THEN
						udiStatus	:= 10022;	//File Close Error While Writing Alarm History
					ELSIF fbFileWrite1.udiStatus = 1914 THEN
						udiStatus	:= 10023;	//Directory Does Not Exist While Writing Alarm History
					ELSE
						udiStatus	:= fbFileWrite1.udiStatus;
					END_IF

				ELSIF fbFileAppend1.udiStatus > 0 AND fbFileAppend1.udiStatus < 65534 THEN
					eStatus		:= Error;

					IF fbFileAppend1.udiStatus = 1900 THEN
						udiStatus	:= 10024;	//File Open Error While Writing Alarm Log
					ELSIF fbFileAppend1.udiStatus = 1901 THEN
						udiStatus	:= 10025;	//File Create Error While Writing Alarm Log
					ELSIF fbFileAppend1.udiStatus = 1913 THEN
						udiStatus	:= 10026;	//Get File Info Error While Writing Alarm Log
					ELSIF fbFileAppend1.udiStatus = 1903 THEN
						udiStatus	:= 10027;	//File Write Error While Writing Alarm Log
					ELSIF fbFileAppend1.udiStatus = 1904 THEN
						udiStatus	:= 10028;	//File Close Error While Writing Alarm Log
					ELSIF fbFileAppend1.udiStatus = 1914 THEN
						udiStatus	:= 10029;	//Directory Does Not Exist While Writing Alarm Log
					ELSE
						udiStatus	:= fbFileAppend1.udiStatus;
					END_IF
				END_IF

			END_IF

		AlarmActResetHistory:
			IF eStatus = Idle OR eStatus = Busy THEN

				eStatus	:= Busy;

				sStatTxt	:= a_sStatText[eStat];

				memset(ADR(a_tyHistoryList) , 0 , SIZEOF(a_tyHistoryList));

				fbFileWrite1(bEn := TRUE);
				IF fbFileWrite1.udiStatus = 0 THEN
					eStatus	:= Done;
				ELSIF fbFileWrite1.udiStatus < 65534 THEN
					eStatus		:= Error;

					IF fbFileWrite1.udiStatus = 1900 THEN
						udiStatus	:= 10030;	//File Open Error While Resetting Alarm History
					ELSIF fbFileWrite1.udiStatus = 1901 THEN
						udiStatus	:= 10031;	//File Create Error While Resetting Alarm History
					ELSIF fbFileWrite1.udiStatus = 1903 THEN
						udiStatus	:= 10032;	//File Write Error While Resetting Alarm History
					ELSIF fbFileWrite1.udiStatus = 1904 THEN
						udiStatus	:= 10033;	//File Close Error While Resetting Alarm History
					ELSIF fbFileWrite1.udiStatus = 1914 THEN
						udiStatus	:= 10034;	//Directory Does Not Exist While Resetting Alarm History
					ELSE
						udiStatus	:= fbFileWrite1.udiStatus;
					END_IF
				END_IF

			END_IF

		AlarmActBGStartLog:
			IF eStatus = Idle OR eStatus = Busy THEN

				sStatTxt	:= a_sStatText[eStat];

				bAlarmLog	:= TRUE;
				eStatus		:= Done;

			END_IF

		AlarmActBGStopLog:
			IF eStatus = Idle OR eStatus = Busy THEN

				sStatTxt	:= a_sStatText[eStat];

				bAlarmLog	:= FALSE;
				eStatus		:= Done;

			END_IF

	END_CASE

END_ACTION
```
